// TwinCAT 3 PLC project MAIN
// ProgramVersion: 3.1.0.9
// CompilerDefines: VISU_USEWSTRING
// libraries:
//   VisuElem3DPath, 3.5.6.0 (System)
//   VisuElemMeter, 3.5.6.0 (System)
//   VisuElems, 3.5.6.10 (System)
//   VisuElemsDateTime, 3.5.6.0 (System)
//   VisuElemsSpecialControls, 3.5.6.0 (System)
//   VisuElemsWinControls, 3.5.6.0 (System)
//   VisuElemTextEditor, 3.5.6.0 (System)
//   visuinputs, 3.5.6.0 (system)
//   VisuNativeControl, 3.5.6.0 (System)
//   Tc2_MC2, * (Beckhoff Automation GmbH)
//   Tc2_NcFifoAxes, * (Beckhoff Automation GmbH)
//   Tc2_Standard, * (Beckhoff Automation GmbH)
//   Tc2_System, * (Beckhoff Automation GmbH)
//   Tc2_Utilities, * (Beckhoff Automation GmbH)
//   Tc3_Interfaces, * (Beckhoff Automation GmbH)
//   Tc3_Module, * (Beckhoff Automation GmbH)
//   VisuDialogs, * (System)
// project tree:
//   DUTs/ ST_CSV_Record.TcDUT
//   / GlobalTextList.TcGTLO, PlcTask.TcTTO, VISU_TASK.TcTTO, 视图管理器.TcVMO (not stored)
//   GVLs/ GVL.TcGVL
//   POUs/ AxisEnable.TcPOU (not stored), AxisMoveAbsoulte.TcPOU, AxisReset.TcPOU, AxisStop.TcPOU, Homing.TcPOU, MAIN.TcPOU, Move_JOG.TcPOU
//   POUs/CSV read_write in text mode/ P_TextModeRead.TcPOU, P_TextModeWrite.TcPOU
//   VISUs/ Visualization.TcVIS
// real-time tasks:
//   TASK PLC_TASK: cycle T#2ms, priority 20, ADS port 350
//   TASK VISU_TASK: cycle T#100000us, priority 30, ADS port 351
//   TASK Kine: cycle T#2ms, priority 21, ADS port 352
// motion (NC):
//   TASK NC-Task 1 SAF: cycle T#2ms, priority 4, ADS port 501
//   TASK NC-Task 1 SVB: cycle T#2ms, priority 8, ADS port 511
//   AXIS Axis 1 (id 1)
//     Dynamic: Acceleration=24000, Deceleration=24000, Jerk=96000
//     Velo: Maximum=6000
//     PositionAreaControl: Enable=false, RefSearch=false
//     TargetPosControl: Enable=false
//     OtherSettings: AllowMotionCmdToSlave=true
//     encoder EncType=19
//       EncPara: ScaleFactorNumerator=0.00274658203125, MaxCount=#xffffffff
//     drive DrvType=16
//       DrvPara: MaxCount=#xffffffff
//         Analog: VeloReferenz=6000
//         TimeComp: TaskDelayCycles=1
//     controller CtrType=1
//       CtrPara: PriorControlFactor=1
//         PosDiffControl: Enable=false
//         Observer: BandWidth=20
//   AXIS Axis 2 (id 2)
//     Dynamic: Acceleration=24000, Deceleration=24000, Jerk=96000
//     Velo: Maximum=6000
//     PositionAreaControl: Enable=false, RefSearch=false
//     TargetPosControl: Enable=false
//     OtherSettings: AllowMotionCmdToSlave=true
//     encoder EncType=19
//       EncPara: ScaleFactorNumerator=0.00274658203125, MaxCount=#xffffffff
//     drive DrvType=16
//       DrvPara: MaxCount=#xffffffff
//         Analog: VeloReferenz=6000
//         TimeComp: TaskDelayCycles=1
//     controller CtrType=1
//       CtrPara: PriorControlFactor=1
//         PosDiffControl: Enable=false
//         Observer: BandWidth=20
//   AXIS Axis 3 (id 3)
//     Dynamic: Acceleration=24000, Deceleration=24000, Jerk=96000
//     Velo: Maximum=6000
//     PositionAreaControl: Enable=false, RefSearch=false
//     TargetPosControl: Enable=false
//     OtherSettings: AllowMotionCmdToSlave=true
//     encoder EncType=19
//       EncPara: ScaleFactorNumerator=0.00274658203125, MaxCount=#xffffffff
//     drive DrvType=16
//       DrvPara: MaxCount=#xffffffff
//         Analog: VeloReferenz=6000
//         TimeComp: TaskDelayCycles=1
//     controller CtrType=1
//       CtrPara: PriorControlFactor=1
//         PosDiffControl: Enable=false
//         Observer: BandWidth=20
//   AXIS Axis 4 (id 4)
//     Dynamic: Acceleration=24000, Deceleration=24000, Jerk=96000
//     Velo: Maximum=6000
//     PositionAreaControl: Enable=false, RefSearch=false
//     TargetPosControl: Enable=false
//     OtherSettings: AllowMotionCmdToSlave=true
//     encoder EncType=19
//       EncPara: ScaleFactorNumerator=0.00274658203125, MaxCount=#xffffffff
//     drive DrvType=16
//       DrvPara: MaxCount=#xffffffff
//         Analog: VeloReferenz=6000
//         TimeComp: TaskDelayCycles=1
//     controller CtrType=1
//       CtrPara: PriorControlFactor=1
//         PosDiffControl: Enable=false
//         Observer: BandWidth=20
//   AXIS Axis 5 (id 5)
//     Dynamic: Acceleration=24000, Deceleration=24000, Jerk=96000
//     Velo: Maximum=6000
//     PositionAreaControl: Enable=false, RefSearch=false
//     TargetPosControl: Enable=false
//     OtherSettings: AllowMotionCmdToSlave=true
//     encoder EncType=19
//       EncPara: ScaleFactorNumerator=0.00274658203125, MaxCount=#xffffffff
//     drive DrvType=16
//       DrvPara: MaxCount=#xffffffff
//         Analog: VeloReferenz=6000
//         TimeComp: TaskDelayCycles=1
//     controller CtrType=1
//       CtrPara: PriorControlFactor=1
//         PosDiffControl: Enable=false
//         Observer: BandWidth=20
//   AXIS Axis 6 (id 6)
//     Dynamic: Acceleration=24000, Deceleration=24000, Jerk=96000
//     Velo: Maximum=6000
//     PositionAreaControl: Enable=false, RefSearch=false
//     TargetPosControl: Enable=false
//     OtherSettings: AllowMotionCmdToSlave=true
//     encoder EncType=19
//       EncPara: ScaleFactorNumerator=0.00274658203125, MaxCount=#xffffffff
//     drive DrvType=16
//       DrvPara: MaxCount=#xffffffff
//         Analog: VeloReferenz=6000
//         TimeComp: TaskDelayCycles=1
//     controller CtrType=1
//       CtrPara: PriorControlFactor=1
//         PosDiffControl: Enable=false
//         Observer: BandWidth=20
// I/O:
//   DEVICE Device 2 (EtherCAT), AmsNetId 192.168.1.1.3.1
//     Box 1 (TOYO NEC-100 Communicator) [TOYO NEC-100 Communicator]
//     Drive 2 (LAN9252-EVB-HBI) [LAN9252-EVB-HBI]
//       modules: Module 1 (csp - axis), Module 2 (csp - axis), Module 3 (csp - axis), Module 4 (csp - axis), Module 5 (csp - axis), Module 6 (csp - axis)
// variable links:
//   NC-Task 1 SAF/Axes/Axis 1 <-> Device 2 (EtherCAT)/Drive 2 (LAN9252-EVB-HBI)
//     Drive/Inputs/In/nState1 <-> Module 6 (csp - axis)/Inputs/Status Word
//     Drive/Inputs/In/nState2 <-> Module 6 (csp - axis)/Inputs/Status Word @bit 8
//     Drive/Outputs/Out/nCtrl1 <-> Module 6 (csp - axis)/Outputs/Control Word
//     Drive/Outputs/Out/nCtrl2 <-> Module 6 (csp - axis)/Outputs/Control Word @bit 8
//     Drive/Outputs/Out/nDataOut1 <-> Module 6 (csp - axis)/Outputs/TargetPosition
//     Enc/Inputs/In/nDataIn1 <-> Module 6 (csp - axis)/Inputs/ActualPosition
//     Enc/Inputs/In/nDcInputTime <-> InfoData/DcInputShift
//   NC-Task 1 SAF/Axes/Axis 2 <-> Device 2 (EtherCAT)/Drive 2 (LAN9252-EVB-HBI)
//     Drive/Inputs/In/nState1 <-> Module 2 (csp - axis)/Inputs/Status Word
//     Drive/Inputs/In/nState2 <-> Module 2 (csp - axis)/Inputs/Status Word @bit 8
//     Drive/Outputs/Out/nCtrl1 <-> Module 2 (csp - axis)/Outputs/Control Word
//     Drive/Outputs/Out/nCtrl2 <-> Module 2 (csp - axis)/Outputs/Control Word @bit 8
//     Drive/Outputs/Out/nDataOut1 <-> Module 2 (csp - axis)/Outputs/TargetPosition
//     Enc/Inputs/In/nDataIn1 <-> Module 2 (csp - axis)/Inputs/ActualPosition
//     Enc/Inputs/In/nDcInputTime <-> InfoData/DcInputShift
//   NC-Task 1 SAF/Axes/Axis 3 <-> Device 2 (EtherCAT)/Drive 2 (LAN9252-EVB-HBI)
//     Drive/Inputs/In/nState1 <-> Module 3 (csp - axis)/Inputs/Status Word
//     Drive/Inputs/In/nState2 <-> Module 3 (csp - axis)/Inputs/Status Word @bit 8
//     Drive/Outputs/Out/nCtrl1 <-> Module 3 (csp - axis)/Outputs/Control Word
//     Drive/Outputs/Out/nCtrl2 <-> Module 3 (csp - axis)/Outputs/Control Word @bit 8
//     Drive/Outputs/Out/nDataOut1 <-> Module 3 (csp - axis)/Outputs/TargetPosition
//     Enc/Inputs/In/nDataIn1 <-> Module 3 (csp - axis)/Inputs/ActualPosition
//     Enc/Inputs/In/nDcInputTime <-> InfoData/DcInputShift
//   NC-Task 1 SAF/Axes/Axis 4 <-> Device 2 (EtherCAT)/Drive 2 (LAN9252-EVB-HBI)
//     Drive/Inputs/In/nState1 <-> Module 4 (csp - axis)/Inputs/Status Word
//     Drive/Inputs/In/nState2 <-> Module 4 (csp - axis)/Inputs/Status Word @bit 8
//     Drive/Outputs/Out/nCtrl1 <-> Module 4 (csp - axis)/Outputs/Control Word
//     Drive/Outputs/Out/nCtrl2 <-> Module 4 (csp - axis)/Outputs/Control Word @bit 8
//     Drive/Outputs/Out/nDataOut1 <-> Module 4 (csp - axis)/Outputs/TargetPosition
//     Enc/Inputs/In/nDataIn1 <-> Module 4 (csp - axis)/Inputs/ActualPosition
//     Enc/Inputs/In/nDcInputTime <-> InfoData/DcInputShift
//   NC-Task 1 SAF/Axes/Axis 5 <-> Device 2 (EtherCAT)/Drive 2 (LAN9252-EVB-HBI)
//     Drive/Inputs/In/nDcOutputTime <-> InfoData/DcOutputShift
//     Drive/Inputs/In/nState1 <-> Module 5 (csp - axis)/Inputs/Status Word
//     Drive/Inputs/In/nState2 <-> Module 5 (csp - axis)/Inputs/Status Word @bit 8
//     Drive/Inputs/In/nState4 @bit 1 <-> WcState/InputToggle
//     Drive/Inputs/In/nState4 <-> WcState/WcState
//     Drive/Outputs/Out/nCtrl1 <-> Module 5 (csp - axis)/Outputs/Control Word
//     Drive/Outputs/Out/nCtrl2 <-> Module 5 (csp - axis)/Outputs/Control Word @bit 8
//     Drive/Outputs/Out/nDataOut1 <-> Module 5 (csp - axis)/Outputs/TargetPosition
//     Enc/Inputs/In/nDataIn1 <-> Module 5 (csp - axis)/Inputs/ActualPosition
//     Enc/Inputs/In/nDcInputTime <-> InfoData/DcInputShift
//     Enc/Inputs/In/nState4 @bit 1 <-> WcState/InputToggle
//     Enc/Inputs/In/nState4 <-> WcState/WcState
//   NC-Task 1 SAF/Axes/Axis 6 <-> Device 2 (EtherCAT)/Drive 2 (LAN9252-EVB-HBI)
//     Drive/Inputs/In/nState1 <-> Module 1 (csp - axis)/Inputs/Status Word
//     Drive/Inputs/In/nState2 <-> Module 1 (csp - axis)/Inputs/Status Word @bit 8
//     Drive/Outputs/Out/nCtrl1 <-> Module 1 (csp - axis)/Outputs/Control Word
//     Drive/Outputs/Out/nCtrl2 <-> Module 1 (csp - axis)/Outputs/Control Word @bit 8
//     Drive/Outputs/Out/nDataOut1 <-> Module 1 (csp - axis)/Outputs/TargetPosition
//     Enc/Inputs/In/nDataIn1 <-> Module 1 (csp - axis)/Inputs/ActualPosition
//     Enc/Inputs/In/nDcInputTime <-> InfoData/DcInputShift
//   MAIN/MAIN Instance <-> Device 2 (EtherCAT)/Box 1 (TOYO NEC-100 Communicator)
//     PlcTask Inputs/MAIN.EcdPos <-> TxPDO/Sa1/EcdPos
//     PlcTask Inputs/MAIN.Status <-> TxPDO/Sa1/Status
//     PlcTask Outputs/MAIN.ABSamount <-> RxPDO/Sa1/ABSamount
//     PlcTask Outputs/MAIN.Control <-> RxPDO/Sa1/Control
//     PlcTask Outputs/MAIN.MovType <-> RxPDO/Sa1/MovType
//   MAIN/MAIN Instance <-> NC-Task 1 SAF/Axes/Axis 1
//     PlcTask Inputs/GVL.Axis[0].NcToPlc <-> Outputs/ToPlc
//     PlcTask Outputs/GVL.Axis[0].PlcToNc <-> Inputs/FromPlc
//   MAIN/MAIN Instance <-> NC-Task 1 SAF/Axes/Axis 2
//     PlcTask Inputs/GVL.Axis[1].NcToPlc <-> Outputs/ToPlc
//     PlcTask Outputs/GVL.Axis[1].PlcToNc <-> Inputs/FromPlc
//   MAIN/MAIN Instance <-> NC-Task 1 SAF/Axes/Axis 3
//     PlcTask Inputs/GVL.Axis[2].NcToPlc <-> Outputs/ToPlc
//     PlcTask Outputs/GVL.Axis[2].PlcToNc <-> Inputs/FromPlc
//   MAIN/MAIN Instance <-> NC-Task 1 SAF/Axes/Axis 4
//     PlcTask Inputs/GVL.Axis[3].NcToPlc <-> Outputs/ToPlc
//     PlcTask Outputs/GVL.Axis[3].PlcToNc <-> Inputs/FromPlc
//   MAIN/MAIN Instance <-> NC-Task 1 SAF/Axes/Axis 5
//     PlcTask Inputs/GVL.Axis[4].NcToPlc <-> Outputs/ToPlc
//     PlcTask Outputs/GVL.Axis[4].PlcToNc <-> Inputs/FromPlc
//   MAIN/MAIN Instance <-> NC-Task 1 SAF/Axes/Axis 6
//     PlcTask Inputs/GVL.Axis[5].NcToPlc <-> Outputs/ToPlc
//     PlcTask Outputs/GVL.Axis[5].PlcToNc <-> Inputs/FromPlc
//   MAIN/MAIN Instance <-> Kinematic/Kinematic_Obj1 (CKineModule)
//     PlcTask Inputs/GVL.ExtPosOK <-> Outputs/ExtPosOK
//     PlcTask Inputs/GVL.ExtPosReady <-> Outputs/ExtPosReady
//     PlcTask Inputs/GVL.ExtPos[{0..5}] <-> Outputs/OutAngle[{0..5}]  (6 links)
//     PlcTask Inputs/GVL.Pos_Now[0] <-> Outputs/Pos_Now[0]
//     PlcTask Inputs/GVL.Pos_Now[1] <-> Outputs/Pos_Now[1]
//     PlcTask Inputs/GVL.Pos_Now[2] <-> Outputs/Pos_Now[2]
//     PlcTask Outputs/GVL.CMoveSpeed <-> Inputs/CSpeed
//     PlcTask Outputs/GVL.KineModuleJob <-> Inputs/KineModlueJob
//     PlcTask Outputs/GVL.LineMoveSpeed <-> Inputs/LineSpeed
//     PlcTask Outputs/GVL.OutActPos[{0..5}] <-> Inputs/InAngle[{5..0}]  (6 links)
//     PlcTask Outputs/GVL.OutCMovePos[0] <-> Inputs/CPos[0]
//     PlcTask Outputs/GVL.OutCMovePos[1] <-> Inputs/CPos[1]
//     PlcTask Outputs/GVL.OutCMovePos[2] <-> Inputs/CPos[2]
//     PlcTask Outputs/GVL.OutMovePos[0] <-> Inputs/InPos[0]
//     PlcTask Outputs/GVL.OutMovePos[1] <-> Inputs/InPos[1]
//     PlcTask Outputs/GVL.OutMovePos[2] <-> Inputs/InPos[2]

CONFIGURATION MAIN
    RESOURCE PLC ON TwinCAT3
        TASK PlcTask(INTERVAL := T#2ms, PRIORITY := 20);
        TASK VISU_TASK(INTERVAL := T#100000us, PRIORITY := 30);
        PROGRAM MAIN WITH PlcTask : MAIN;
        PROGRAM VisuElems_Visu_Prg WITH VISU_TASK : VisuElems.Visu_Prg;
    END_RESOURCE
END_CONFIGURATION

// ---- DUTs/ST_CSV_Record.TcDUT
TYPE ST_CSV_Record :
STRUCT
	sName 	: T_MaxString 	:= '';
	nNumber	: UDINT 		:= 0;
	fPos	: LREAL 		:= 0.0;
	bOP		: BOOL 			:= FALSE;
	sDesc	: STRING(40)	:= '';
	data	: ARRAY[0..7] OF BYTE;
END_STRUCT
END_TYPE

// ---- GVLs/GVL.TcGVL
VAR_GLOBAL CONSTANT
	MAX_CSV_ROWS 			: UDINT := 1;//1680;//hang
	MAX_CSV_COLUMNS 		: UDINT := 3;//lie 0-5
	MAX_CSV_FIELD_LENGTH	: UDINT := 20;
END_VAR

VAR_GLOBAL

axisNum: INT:=0;
//Axis Bind link
Axis:ARRAY[0..5]OF AXIS_REF;	

//Axis Power On
AxisPower:ARRAY[0..5]OF MC_Power;
AxisPowerTrigger:ARRAY[0..5]OF BOOL;
AxisPowerReady:ARRAY[0..5]OF BOOL;
AxisPowerBusy:ARRAY[0..5]OF BOOL;
AxisPowerActive:ARRAY[0..5]OF BOOL;
AxisPowerError:ARRAY[0..5]OF BOOL;
AxisPowerErrorID:ARRAY[0..5]OF UDINT;

//Axis Move Absolute
AxisMoveAbsolute:ARRAY[0..5]OF MC_MoveAbsolute;
AxisMoveTrigger:ARRAY[0..5]OF BOOL;
AxisMovePosition:ARRAY[0..5]OF LREAL;
AxisMoveSpeed:ARRAY[0..5]OF LREAL;
AxisMoveAcceleration:ARRAY[0..5]OF LREAL;
AxisMoveDeceleration:ARRAY[0..5]OF LREAL;
AxisMoveJerk:ARRAY[0..5]OF LREAL;
AxisMoveAbsoluteDone:ARRAY[0..5]OF BOOL;
AxisMoveAbsoluteBusy:ARRAY[0..5]OF BOOL;
AxisMoveAbsoluteActive:ARRAY[0..5]OF BOOL;
AxisMoveAbsoluteCommandAborted:ARRAY[0..5]OF BOOL;
AxisMoveAbsoluteError:ARRAY[0..5]OF BOOL;
AxisMoveAbsoluteErrorID:ARRAY[0..5]OF UDINT;

//Axis Stop
MC_Stop1:ARRAY[0..5]OF MC_Stop;
AxisStopTrigger:ARRAY[0..5]OF BOOL;
AxisStopDeceleration:ARRAY[0..5]OF LREAL;
AxisStopJerk:ARRAY[0..5]OF LREAL;
AxisStopDone:ARRAY[0..5]OF BOOL;
AxisStopBusy:ARRAY[0..5]OF BOOL;
AxisStopActive:ARRAY[0..5]OF BOOL;
AxisStopCommandAborted:ARRAY[0..5]OF BOOL;
AxisStopError:ARRAY[0..5]OF BOOL;
AxisStopErrorID:ARRAY[0..5]OF UDINT;

//MoveJOG
MoveJOG:ARRAY[0..5]OF MC_Jog;
JogFw:ARRAY[0..5]OF BOOL;
JogBw:ARRAY[0..5]OF BOOL;
JogMode:ARRAY[0..5]OF E_JogMode;
JogPosition:ARRAY[0..5]OF LREAL;
Jogvelocity:ARRAY[0..5]OF LREAL;
JogAcceleration:ARRAY[0..5]OF LREAL;
JogDeceleration:ARRAY[0..5]OF LREAL;
JogJerk:ARRAY[0..5]OF LREAL;
JogDone:ARRAY[0..5]OF BOOL;
JogBusy:ARRAY[0..5]OF BOOL;
JogActive:ARRAY[0..5]OF BOOL;
JogCommandAborted:ARRAY[0..5]OF BOOL;
JogError:ARRAY[0..5]OF BOOL;
JogErrorID:ARRAY[0..5]OF UDINT;

//Reset
MC_Resrt_0: ARRAY[0..5] OF MC_Reset;
AxisResetDone: ARRAY[0..5] OF BOOL;
AxisResetTrigger: ARRAY[0..5] OF BOOL;
AxisResetBusy: ARRAY[0..5] OF BOOL;
AxisResetError: ARRAY[0..5] OF BOOL;
AxisResetErrorID: ARRAY[0..5] OF UDINT;

//HOME
home_1: ARRAY[0..5] OF MC_HOME;
Home_Done: ARRAY[0..5] OF BOOL;
Home: ARRAY[0..5] OF BOOL;
Home_Pos: ARRAY[0..5] OF LREAL;
Home_Mode: ARRAY[0..5] OF MC_HomingMode;
Home_cal: ARRAY[0..5] OF BOOL;
Home_busy: ARRAY[0..5] OF BOOL;
Home_Active: ARRAY[0..5] OF BOOL;
Home_CommandAborted: ARRAY[0..5] OF BOOL;
Home_Error: ARRAY[0..5] OF BOOL;
Home_ErrorID: ARRAY[0..5] OF UDINT;
	
MoveA:ARRAY [0..5] OF LREAL;
MoveAString:ARRAY [0..5] OF STRING := ['0','0','0','0','0','0'];

FIFO_POS AT%I*:ARRAY[0..5]OF LREAL;//来自ros的外部位置
ExtPos AT%I*:ARRAY[0..5]OF LREAL;//来自CPPModule的外部位置
ExtPosOK AT%I*:BOOL;//外部位置执行结束标志
ExtPosReady AT%I*:BOOL;//外部位置规划完成
OutActPos AT%Q*:ARRAY[0..5]OF LREAL;//给CPPModule的实时位置

OutMovePos AT%Q*:ARRAY[0..2]OF LREAL;//直线规划增量
OutMovePosString:ARRAY[0..2]OF STRING := ['0','0','-0.1'];//增量字符串值
LineMoveSpeed AT%Q*:LREAL;//运动速度
LineMoveSpeedString:STRING:='0.05';

OutCMovePos AT%Q*:ARRAY[0..2]OF LREAL;//笛卡尔规划增量
OutCMovePosString:ARRAY[0..2]OF STRING := ['0.4','0.2','0.2'];//增量字符串值
CMoveSpeed AT%Q*:LREAL;//运动速度
CMoveSpeedString:STRING:='0.3';

KineModuleJob AT%Q*:INT:=0;//CPPModule状态机控制
Pos_Now AT%I*:ARRAY[0..2]OF LREAL;//CPPModule输出实时笛卡尔坐标
END_VAR

// ---- POUs/MAIN.TcPOU
PROGRAM MAIN
VAR
bChangeSeparatorToComma	: BOOL := TRUE;
P_TextModeWrite_WriteTrigger:BOOL:=FALSE;
P_TextModeWrite_WriteFilePath:T_MaxString := 'C:\Users\Administrator\Desktop\Pos.csv';
P_TextModeRead_ReadTrigger:BOOL:=FALSE;
P_TextModeRead_ReadFilePath:T_MaxString := 'C:\Users\Administrator\Desktop\Pos.csv';

CurrentJob: INT:= 0;//Job Code
CurrentJobState:STRING(80);//Say in which state

LAMP:BOOL;
POWER:BOOL;
Move_AB:BOOL;

SetPointGenEnable:ARRAY [0..5] OF MC_ExtSetPointGenEnable;
SetpointGenDisable:ARRAY [0..5] OF MC_ExtSetpointGenDisable;
SetPointGenEnable_output: ARRAY [0..5] OF ST_McOutputs;
SetPointGenDisable_output: ARRAY [0..5] OF ST_McOutputs;
enable:ARRAY [0..5] OF BOOL;
disable:ARRAY [0..5] OF BOOL;

position:ARRAY [0..5] OF LREAL;
velocity:ARRAY [0..5] OF LREAL;
direction:ARRAY [0..5] OF DINT;
acceleration:ARRAY [0..5] OF LREAL;

Pos_arr1:ARRAY[0..4999,0..5] OF LREAL;
i:INT;
FiFo_GetDimension: FiFoGetDimension;
fifo_display: STRING(255);

FiFo_GroupIntegrate1,FiFo_GroupIntegrate2,FiFo_GroupIntegrate3,FiFo_GroupIntegrate4,FiFo_GroupIntegrate6,FiFo_GroupIntegrate5: FiFoGroupIntegrate;
FiFo_SetChannelOverride:FiFoSetChannelOverride;
FiFo_Groupout1,FiFo_Groupout2,FiFo_Groupout3,FiFo_Groupout4,FiFo_Groupout5,FiFo_Groupout6,FiFo_Disintegrate,FiFo_Override_output:st_mcoutputs;
integrate_do:BOOL;
FiFo_GroupDisintegrate:FiFoGroupDisintegrate;

FiFo_Start:FiFoStart;
start_do:BOOL;
FiFo_Stop:FiFoStop;
stop_do:BOOL;
fifo_startoutput,fifo_stopoutput:st_mcoutputs;

FiFo_Write:FiFoWrite;
FIFO_write_do:BOOL;
FiFo_overWrite:FiFoOverwrite;
FIFO_overwrite_do:BOOL;
FIFO_write_output:st_mcoutputs;

END_VAR
VAR CONSTANT
	GlobalSetSpeed : ARRAY[0..5]OF LREAL:=[3200,3200,3200,3200,3200,3200];
END_VAR

IF bChangeSeparatorToComma THEN
	DEFAULT_CSV_FIELD_SEP := 16#2C;(* Comma ASCII code *)
ELSE
	DEFAULT_CSV_FIELD_SEP := 16#3B;(* Semicolon ASCII code *)
END_IF

IF FiFo_GetDimension.iNoOfAxes=6 AND FiFo_GetDimension.iNoOfFifoEntries=200 THEN
	fifo_display:='Parameters OK';
ELSE
	fifo_display:='Parameters Bad';
END_IF

//fifo();

GVL.LineMoveSpeed:=STRING_TO_LREAL(GVL.LineMoveSpeedString);
GVL.CMoveSpeed:=STRING_TO_LREAL(GVL.CMoveSpeedString);
GVL.OutMovePos[0]:=STRING_TO_LREAL(GVL.OutMovePosString[0]);
GVL.OutMovePos[1]:=STRING_TO_LREAL(GVL.OutMovePosString[1]);
GVL.OutMovePos[2]:=STRING_TO_LREAL(GVL.OutMovePosString[2]);
GVL.OutCMovePos[0]:=STRING_TO_LREAL(GVL.OutCMovePosString[0]);
GVL.OutCMovePos[1]:=STRING_TO_LREAL(GVL.OutCMovePosString[1]);
GVL.OutCMovePos[2]:=STRING_TO_LREAL(GVL.OutCMovePosString[2]);
GVL.MoveA[0]:=STRING_TO_LREAL(GVL.MoveAString[0])*24.995;
GVL.MoveA[1]:=STRING_TO_LREAL(GVL.MoveAString[1])*32.28;
GVL.MoveA[2]:=STRING_TO_LREAL(GVL.MoveAString[2])*49.845;
GVL.MoveA[3]:=STRING_TO_LREAL(GVL.MoveAString[3])*50.905;
GVL.MoveA[4]:=STRING_TO_LREAL(GVL.MoveAString[4])*80.34;
GVL.MoveA[5]:=STRING_TO_LREAL(GVL.MoveAString[5])*60.5;
GVL.OutActPos[0]:=-GVL.Axis[0].NcToPlc.ActPos/24.995;
GVL.OutActPos[1]:=-GVL.Axis[1].NcToPlc.ActPos/32.28;
GVL.OutActPos[2]:=GVL.Axis[2].NcToPlc.ActPos/49.845;
GVL.OutActPos[3]:=GVL.Axis[3].NcToPlc.ActPos/50.905;
GVL.OutActPos[4]:=GVL.Axis[4].NcToPlc.ActPos/80.34;
GVL.OutActPos[5]:=GVL.Axis[5].NcToPlc.ActPos/60.5;

IF GVL.ExtPosReady = FALSE THEN	
MC_ExtSetPointGenFeed(Position:=-GVL.OutActPos[0]*24.995,Velocity:= 0,Acceleration:=0,Direction:=1,Axis:=Axis[0]);	
MC_ExtSetPointGenFeed(Position:=-GVL.OutActPos[1]*32.28,Velocity:= 0,Acceleration:=0,Direction:=1,Axis:=Axis[1]);		
MC_ExtSetPointGenFeed(Position:=GVL.OutActPos[2]*49.845,Velocity:= 0,Acceleration:=0,Direction:=1,Axis:=Axis[2]);		
MC_ExtSetPointGenFeed(Position:=GVL.OutActPos[3]*50.905,Velocity:= 0,Acceleration:=0,Direction:=1,Axis:=Axis[3]);		
MC_ExtSetPointGenFeed(Position:=GVL.OutActPos[4]*80.34,Velocity:= 0,Acceleration:=0,Direction:=1,Axis:=Axis[4]);		
MC_ExtSetPointGenFeed(Position:=GVL.OutActPos[5]*60.5,Velocity:= 0,Acceleration:=0,Direction:=1,Axis:=Axis[5]);		
END_IF

CASE CurrentJob OF	
	0://None state
		AxisStopTrigger[0]:=FALSE;AxisStopTrigger[1]:=FALSE;AxisStopTrigger[2]:=FALSE;
		AxisStopTrigger[3]:=FALSE;AxisStopTrigger[4]:=FALSE;AxisStopTrigger[5]:=FALSE;
		AxisStop();//失能功能块
		
		JogFw[0]:=FALSE;JogFw[1]:=FALSE;JogFw[2]:=FALSE;JogFw[3]:=FALSE;JogFw[4]:=FALSE;JogFw[5]:=FALSE;
		JogBw[0]:=FALSE;JogBw[1]:=FALSE;JogBw[2]:=FALSE;JogBw[3]:=FALSE;JogBw[4]:=FALSE;JogBw[5]:=FALSE;
		Move_JOG();//失能功能块
		
		AxisMoveTrigger[0]:=FALSE;AxisMoveTrigger[1]:=FALSE;AxisMoveTrigger[2]:=FALSE;
		AxisMoveTrigger[3]:=FALSE;AxisMoveTrigger[4]:=FALSE;AxisMoveTrigger[5]:=FALSE;
		AxisMoveAbsoulte();//失能功能块
		
		Home[0]:=FALSE;Home[1]:=FALSE;Home[2]:=FALSE;
		Home[3]:=FALSE;Home[4]:=FALSE;Home[5]:=FALSE;
		Homing();//失能功能块	

		AxisResetTrigger[0]:=FALSE;AxisResetTrigger[1]:=FALSE;AxisResetTrigger[2]:=FALSE;
		AxisResetTrigger[3]:=FALSE;AxisResetTrigger[4]:=FALSE;AxisResetTrigger[5]:=FALSE;
		AxisReset();//失能功能块
		
		P_TextModeWrite_WriteTrigger:=FALSE;
		P_TextModeWrite();	
		P_TextModeRead_ReadTrigger:=FALSE;
		P_TextModeRead();//失能功能块
		
		SetPointGenEnable[0].Execute:=FALSE;SetPointGenEnable[1].Execute:=FALSE;
		SetPointGenEnable[2].Execute:=FALSE;SetPointGenEnable[3].Execute:=FALSE;
		SetPointGenEnable[4].Execute:=FALSE;SetPointGenEnable[5].Execute:=FALSE;

		SetPointGenDisable[0].Execute:=FALSE;SetPointGenDisable[1].Execute:=FALSE;		
		SetPointGenDisable[2].Execute:=FALSE;SetPointGenDisable[3].Execute:=FALSE;		
		SetPointGenDisable[4].Execute:=FALSE;SetPointGenDisable[5].Execute:=FALSE;		
		setpositionGen();
		
		JogMode[0]:=MC_JOGMODE_STANDARD_FAST;
		JogMode[1]:=MC_JOGMODE_STANDARD_FAST;
		JogMode[2]:=MC_JOGMODE_STANDARD_FAST;
		JogMode[3]:=MC_JOGMODE_STANDARD_FAST;
		JogMode[4]:=MC_JOGMODE_STANDARD_FAST;
		JogMode[5]:=MC_JOGMODE_STANDARD_FAST;

		GVL.KineModuleJob:=0;
	
		CurrentJobState:='Wait Command';
		i:=0;
	1://SetZero
		Home[0]:=TRUE;Home[1]:=TRUE;Home[2]:=TRUE;
		Home[3]:=TRUE;Home[4]:=TRUE;Home[5]:=TRUE;
		Home_Mode[0]:=MC_Direct;Home_Mode[1]:=MC_Direct;Home_Mode[2]:=MC_Direct;
		Home_Mode[3]:=MC_Direct;Home_Mode[4]:=MC_Direct;Home_Mode[5]:=MC_Direct;
		Home_Pos[0]:=0;Home_Pos[1]:=0;Home_Pos[2]:=0;
		Home_Pos[3]:=0;Home_Pos[4]:=0;Home_Pos[5]:=0;
		Homing();

		IF Home_Done[0]=TRUE AND 
		   Home_Done[1]=TRUE AND 
		   Home_Done[2]=TRUE AND 
		   Home_Done[3]=TRUE AND 
		   Home_Done[4]=TRUE AND 
		   Home_Done[5]=TRUE THEN
			CurrentJob:=0;
			CurrentJobState:='Set Origin Done!';
		ELSE
			CurrentJobState:='Set Origin Doing';
		END_IF
	2://直线插补
		setpointgenenable[0].Execute:=TRUE;setpointgenenable[1].Execute:=TRUE;
		setpointgenenable[2].Execute:=TRUE;setpointgenenable[3].Execute:=TRUE;
		setpointgenenable[4].Execute:=TRUE;setpointgenenable[5].Execute:=TRUE;
		IF  SetPointGenEnable[0].Enabled AND
			SetPointGenEnable[1].Enabled AND
			SetPointGenEnable[2].Enabled AND
			SetPointGenEnable[3].Enabled AND
			SetPointGenEnable[4].Enabled AND
			SetPointGenEnable[5].Enabled THEN

			//IF(GVL.ExtPosOK = TRUE) THEN
			IF i > 4998 THEN
				SetPointGenDisable[0].Execute:=TRUE;SetPointGenDisable[1].Execute:=TRUE;
				SetPointGenDisable[2].Execute:=TRUE;SetPointGenDisable[3].Execute:=TRUE;
				SetPointGenDisable[4].Execute:=TRUE;SetPointGenDisable[5].Execute:=TRUE;
				setpositionGen();
				CurrentJob:=0;
			ELSE
				i:=i+1;
		
				MC_ExtSetPointGenFeed(Position:=Pos_arr1[i,0]*24.995,Velocity:= 0,Acceleration:=0,Direction:=1,Axis:=Axis[0]);
			
				MC_ExtSetPointGenFeed(Position:=Pos_arr1[i,1]*32.28,Velocity:= 0,Acceleration:=0,Direction:=1,Axis:=Axis[1]);
			
				MC_ExtSetPointGenFeed(Position:=Pos_arr1[i,2]*49.845,Velocity:= 0,Acceleration:=0,Direction:=1,Axis:=Axis[2]);
			
				MC_ExtSetPointGenFeed(Position:=Pos_arr1[i,3]*50.905,Velocity:= 0,Acceleration:=0,Direction:=1,Axis:=Axis[3]);
			
				MC_ExtSetPointGenFeed(Position:=Pos_arr1[i,4]*80.34,Velocity:= 0,Acceleration:=0,Direction:=1,Axis:=Axis[4]);
			
				MC_ExtSetPointGenFeed(Position:=Pos_arr1[i,5]*60.5,Velocity:= 0,Acceleration:=0,Direction:=1,Axis:=Axis[5]);
			END_IF
			//GVL.KineModuleJob:=4;
			//IF GVL.ExtPosReady THEN
			//MC_ExtSetPointGenFeed(Position:=-ExtPos[0]*24.995,Velocity:= 0,Acceleration:=0,Direction:=1,Axis:=Axis[0]);
			
			//MC_ExtSetPointGenFeed(Position:=-ExtPos[1]*32.28,Velocity:= 0,Acceleration:=0,Direction:=1,Axis:=Axis[1]);
			
			//MC_ExtSetPointGenFeed(Position:=ExtPos[2]*49.845,Velocity:= 0,Acceleration:=0,Direction:=1,Axis:=Axis[2]);
			
			//MC_ExtSetPointGenFeed(Position:=ExtPos[3]*50.905,Velocity:= 0,Acceleration:=0,Direction:=1,Axis:=Axis[3]);
			
			//MC_ExtSetPointGenFeed(Position:=ExtPos[4]*80.34,Velocity:= 0,Acceleration:=0,Direction:=1,Axis:=Axis[4]);
			
			//MC_ExtSetPointGenFeed(Position:=ExtPos[5]*60.5,Velocity:= 0,Acceleration:=0,Direction:=1,Axis:=Axis[5]);		
			//END_IF
		END_IF
		setpositionGen();
	3://JogForward
		JogFw[axisNum]:=TRUE;
		Move_JOG();
		CurrentJob:=3;
		CurrentJobState:='Jog Forward';
	4://JogBackward
		JogBw[axisNum]:=TRUE;
		Move_JOG();
		CurrentJob:=4;
		CurrentJobState:='Jog Backward';
	5://Stop
		AxisStopDeceleration[0]:=15000;AxisStopDeceleration[1]:=15000;AxisStopDeceleration[2]:=15000;
		AxisStopDeceleration[3]:=15000;AxisStopDeceleration[4]:=15000;AxisStopDeceleration[5]:=15000;
		AxisStopTrigger[0]:=TRUE;AxisStopTrigger[1]:=TRUE;AxisStopTrigger[2]:=TRUE;
		AxisStopTrigger[3]:=TRUE;AxisStopTrigger[4]:=TRUE;AxisStopTrigger[5]:=TRUE;
		AxisStop();
		IF AxisStopDone[0]=TRUE AND
		   AxisStopDone[1]=TRUE AND
		   AxisStopDone[2]=TRUE AND
		   AxisStopDone[3]=TRUE AND
		   AxisStopDone[4]=TRUE AND
		   AxisStopDone[5]=TRUE THEN
			CurrentJobState:='Stop Done';
			CurrentJob:=0;
		ELSE
			CurrentJobState:='Stop Doing';
		END_IF
	6://Move To HOME
		AxisMovePosition[0]:=-3683.8943;AxisMovePosition[1]:=5173.9531;AxisMovePosition[2]:=318.8809;
		AxisMovePosition[3]:=5194.3991;AxisMovePosition[4]:=307.0219;AxisMovePosition[5]:=774.2587;	
		AxisMoveSpeed[0]:=2000;AxisMoveSpeed[1]:=2000;AxisMoveSpeed[2]:=2000;
		AxisMoveSpeed[3]:=2000;AxisMoveSpeed[4]:=2000;AxisMoveSpeed[5]:=2000;
		
		AxisMoveTrigger[0]:=TRUE;AxisMoveTrigger[1]:=TRUE;AxisMoveTrigger[2]:=TRUE;
		AxisMoveTrigger[3]:=TRUE;AxisMoveTrigger[4]:=TRUE;AxisMoveTrigger[5]:=TRUE;
		AxisMoveAbsoulte();
		
		IF AxisMoveAbsoluteDone[0]=TRUE AND 
		   AxisMoveAbsoluteDone[1]=TRUE AND 
		   AxisMoveAbsoluteDone[2]=TRUE AND 
		   AxisMoveAbsoluteDone[3]=TRUE AND 
		   AxisMoveAbsoluteDone[4]=TRUE AND 
		   AxisMoveAbsoluteDone[5]=TRUE THEN			
			CurrentJobState:='Home Done';
			CurrentJob:=1;			
		ELSE
			CurrentJobState:='Home Doing';
		END_IF
	7://Move To A
		AxisMovePosition[0]:=MoveA[0];AxisMovePosition[1]:=MoveA[1];AxisMovePosition[2]:=MoveA[2];
		AxisMovePosition[3]:=MoveA[3];AxisMovePosition[4]:=MoveA[4];AxisMovePosition[5]:=MoveA[5];
		
		AxisMoveSpeed[0]:=GlobalSetSpeed[0];AxisMoveSpeed[1]:=GlobalSetSpeed[1];AxisMoveSpeed[2]:=GlobalSetSpeed[2];
		AxisMoveSpeed[3]:=GlobalSetSpeed[3];AxisMoveSpeed[4]:=GlobalSetSpeed[4];AxisMoveSpeed[5]:=GlobalSetSpeed[5];
		
		AxisMoveTrigger[0]:=TRUE;AxisMoveTrigger[1]:=TRUE;AxisMoveTrigger[2]:=TRUE;
		AxisMoveTrigger[3]:=TRUE;AxisMoveTrigger[4]:=TRUE;AxisMoveTrigger[5]:=TRUE;
		AxisMoveAbsoulte();
		
		IF AxisMoveAbsoluteDone[0]=TRUE AND 
		   AxisMoveAbsoluteDone[1]=TRUE AND 
		   AxisMoveAbsoluteDone[2]=TRUE AND 
		   AxisMoveAbsoluteDone[3]=TRUE AND 
		   AxisMoveAbsoluteDone[4]=TRUE AND 
		   AxisMoveAbsoluteDone[5]=TRUE THEN		
			CurrentJobState:='MOVE A Done';
			CurrentJob:=0;		
		ELSE
			CurrentJobState:='MOVE A Doing';
		END_IF
	8://往复运动
		IF Move_AB=FALSE THEN
		//AxisMovePosition[0]:=-742579.6646;AxisMovePosition[1]:=5125.997925;AxisMovePosition[2]:=223.8519;
		//AxisMovePosition[3]:=5161.5829;AxisMovePosition[4]:=-31.9675;AxisMovePosition[5]:=774.2587;	
		AxisMovePosition[0]:=0;AxisMovePosition[1]:=0;AxisMovePosition[2]:=0;
		AxisMovePosition[3]:=0;AxisMovePosition[4]:=0;AxisMovePosition[5]:=0;
		ELSE
		AxisMovePosition[0]:=MoveA[0];AxisMovePosition[1]:=MoveA[1];AxisMovePosition[2]:=MoveA[2];
		AxisMovePosition[3]:=MoveA[3];AxisMovePosition[4]:=MoveA[4];AxisMovePosition[5]:=MoveA[5];	
		END_IF
		AxisMoveSpeed[0]:=2000;AxisMoveSpeed[1]:=2000;AxisMoveSpeed[2]:=2000;
		AxisMoveSpeed[3]:=2000;AxisMoveSpeed[4]:=2000;AxisMoveSpeed[5]:=2000;
		
		AxisMoveTrigger[0]:=TRUE;AxisMoveTrigger[1]:=TRUE;AxisMoveTrigger[2]:=TRUE;
		AxisMoveTrigger[3]:=TRUE;AxisMoveTrigger[4]:=TRUE;AxisMoveTrigger[5]:=TRUE;
		AxisMoveAbsoulte();
		
		IF AxisMoveAbsoluteDone[0]=TRUE AND 
		   AxisMoveAbsoluteDone[1]=TRUE AND 
		   AxisMoveAbsoluteDone[2]=TRUE AND 
		   AxisMoveAbsoluteDone[3]=TRUE AND 
		   AxisMoveAbsoluteDone[4]=TRUE AND 
		   AxisMoveAbsoluteDone[5]=TRUE THEN	
		   Move_AB:= NOT Move_AB;
		   AxisMoveTrigger[0]:=FALSE;AxisMoveTrigger[1]:=FALSE;AxisMoveTrigger[2]:=FALSE;
		   AxisMoveTrigger[3]:=FALSE;AxisMoveTrigger[4]:=FALSE;AxisMoveTrigger[5]:=FALSE;
		   AxisMoveAbsoulte();//失能功能块
		END_IF
		CurrentJobState:='Reciprocating Doing';
	9://复位
		AxisResetTrigger[0]:=TRUE;AxisResetTrigger[1]:=TRUE;AxisResetTrigger[2]:=TRUE;
		AxisResetTrigger[3]:=TRUE;AxisResetTrigger[4]:=TRUE;AxisResetTrigger[5]:=TRUE;
		AxisReset();
		IF AxisResetDone[0]=TRUE AND
		   AxisResetDone[1]=TRUE AND
		   AxisResetDone[2]=TRUE AND
		   AxisResetDone[3]=TRUE AND
		   AxisResetDone[4]=TRUE AND
		   AxisResetDone[5]=TRUE THEN	
			CurrentJobState:='Axis Reset Done';
			CurrentJob:=0;
		ELSE
			CurrentJobState:='Axis Reset Doing';
		END_IF
	10://read csv
		//P_TextModeRead_ReadTrigger:=TRUE;
		//CurrentJobState:='Read CSV';
		//P_TextModeRead();
		GVL.KineModuleJob:=2;
		CurrentJob:=0;
	11://Move to origin
		AxisMovePosition[0]:=0;AxisMovePosition[1]:=0;AxisMovePosition[2]:=0;
		AxisMovePosition[3]:=0;AxisMovePosition[4]:=0;AxisMovePosition[5]:=0;
		
		AxisMoveSpeed[0]:=2000;AxisMoveSpeed[1]:=2000;AxisMoveSpeed[2]:=2000;
		AxisMoveSpeed[3]:=2000;AxisMoveSpeed[4]:=2000;AxisMoveSpeed[5]:=2000;
		
		AxisMoveTrigger[0]:=TRUE;AxisMoveTrigger[1]:=TRUE;AxisMoveTrigger[2]:=TRUE;
		AxisMoveTrigger[3]:=TRUE;AxisMoveTrigger[4]:=TRUE;AxisMoveTrigger[5]:=TRUE;
		AxisMoveAbsoulte();
		
		IF AxisMoveAbsoluteDone[0]=TRUE AND 
		   AxisMoveAbsoluteDone[1]=TRUE AND 
		   AxisMoveAbsoluteDone[2]=TRUE AND 
		   AxisMoveAbsoluteDone[3]=TRUE AND 
		   AxisMoveAbsoluteDone[4]=TRUE AND 
		   AxisMoveAbsoluteDone[5]=TRUE THEN		
			CurrentJobState:='MOVE Origin Done';
			CurrentJob:=0;		
		ELSE
			CurrentJobState:='MOVE Origin Doing';
		END_IF
	12://直线插补
		setpointgenenable[0].Execute:=TRUE;setpointgenenable[1].Execute:=TRUE;
		setpointgenenable[2].Execute:=TRUE;setpointgenenable[3].Execute:=TRUE;
		setpointgenenable[4].Execute:=TRUE;setpointgenenable[5].Execute:=TRUE;
		IF  SetPointGenEnable[0].Enabled AND
			SetPointGenEnable[1].Enabled AND
			SetPointGenEnable[2].Enabled AND
			SetPointGenEnable[3].Enabled AND
			SetPointGenEnable[4].Enabled AND
			SetPointGenEnable[5].Enabled THEN
			
			IF(GVL.ExtPosOK = TRUE) THEN			
				SetPointGenDisable[0].Execute:=TRUE;SetPointGenDisable[1].Execute:=TRUE;
				SetPointGenDisable[2].Execute:=TRUE;SetPointGenDisable[3].Execute:=TRUE;
				SetPointGenDisable[4].Execute:=TRUE;SetPointGenDisable[5].Execute:=TRUE;
				setpositionGen();
				CurrentJob:=0;
			END_IF
			
			GVL.KineModuleJob:=3;
			IF GVL.ExtPosReady THEN
			MC_ExtSetPointGenFeed(Position:=ExtPos[0]*24.995,Velocity:= 0,Acceleration:=0,Direction:=1,Axis:=Axis[0]);
			
			MC_ExtSetPointGenFeed(Position:=-ExtPos[1]*32.28,Velocity:= 0,Acceleration:=0,Direction:=1,Axis:=Axis[1]);
			
			MC_ExtSetPointGenFeed(Position:=ExtPos[2]*49.845,Velocity:= 0,Acceleration:=0,Direction:=1,Axis:=Axis[2]);
			
			MC_ExtSetPointGenFeed(Position:=ExtPos[3]*50.905,Velocity:= 0,Acceleration:=0,Direction:=1,Axis:=Axis[3]);
			
			MC_ExtSetPointGenFeed(Position:=ExtPos[4]*80.34,Velocity:= 0,Acceleration:=0,Direction:=1,Axis:=Axis[4]);
			
			MC_ExtSetPointGenFeed(Position:=ExtPos[5]*60.5,Velocity:= 0,Acceleration:=0,Direction:=1,Axis:=Axis[5]);		
			END_IF
		END_IF
		setpositionGen();
	13://关节空间运动
		GVL.KineModuleJob:=1;
		CurrentJob:=0;
END_CASE

//错误检测
IF  AxisPowerError[0] OR
	AxisPowerError[1] OR
	AxisPowerError[2] OR
	AxisPowerError[3] OR
	AxisPowerError[4] OR
	AxisPowerError[5] THEN
	//POWER:=FALSE;
	CurrentJob:=9;
END_IF
//电机上下电
IF POWER=TRUE THEN
	AxisPowerTrigger[0]:=TRUE;
	AxisPowerTrigger[1]:=TRUE;
	AxisPowerTrigger[2]:=TRUE;
	AxisPowerTrigger[3]:=TRUE;
	AxisPowerTrigger[4]:=TRUE;
	AxisPowerTrigger[5]:=TRUE;
	AxisEnable();
	IF  AxisPowerReady[0]=TRUE AND 
		AxisPowerReady[1]=TRUE AND 
		AxisPowerReady[2]=TRUE AND 
		AxisPowerReady[3]=TRUE AND
		AxisPowerReady[4]=TRUE AND 
		AxisPowerReady[5]=TRUE THEN
		LAMP:=TRUE;
	END_IF
ELSE
	AxisPowerTrigger[0]:=FALSE;
	AxisPowerTrigger[1]:=FALSE;
	AxisPowerTrigger[2]:=FALSE;
	AxisPowerTrigger[3]:=FALSE;
	AxisPowerTrigger[4]:=FALSE;
	AxisPowerTrigger[5]:=FALSE;
	AxisEnable();
	IF  AxisPowerReady[0]=FALSE AND
		AxisPowerReady[1]=FALSE AND
		AxisPowerReady[2]=FALSE AND
		AxisPowerReady[3]=FALSE AND
		AxisPowerReady[4]=FALSE AND
		AxisPowerReady[5]=FALSE THEN
		LAMP:=FALSE;   
	END_IF
END_IF

ACTION fifo:
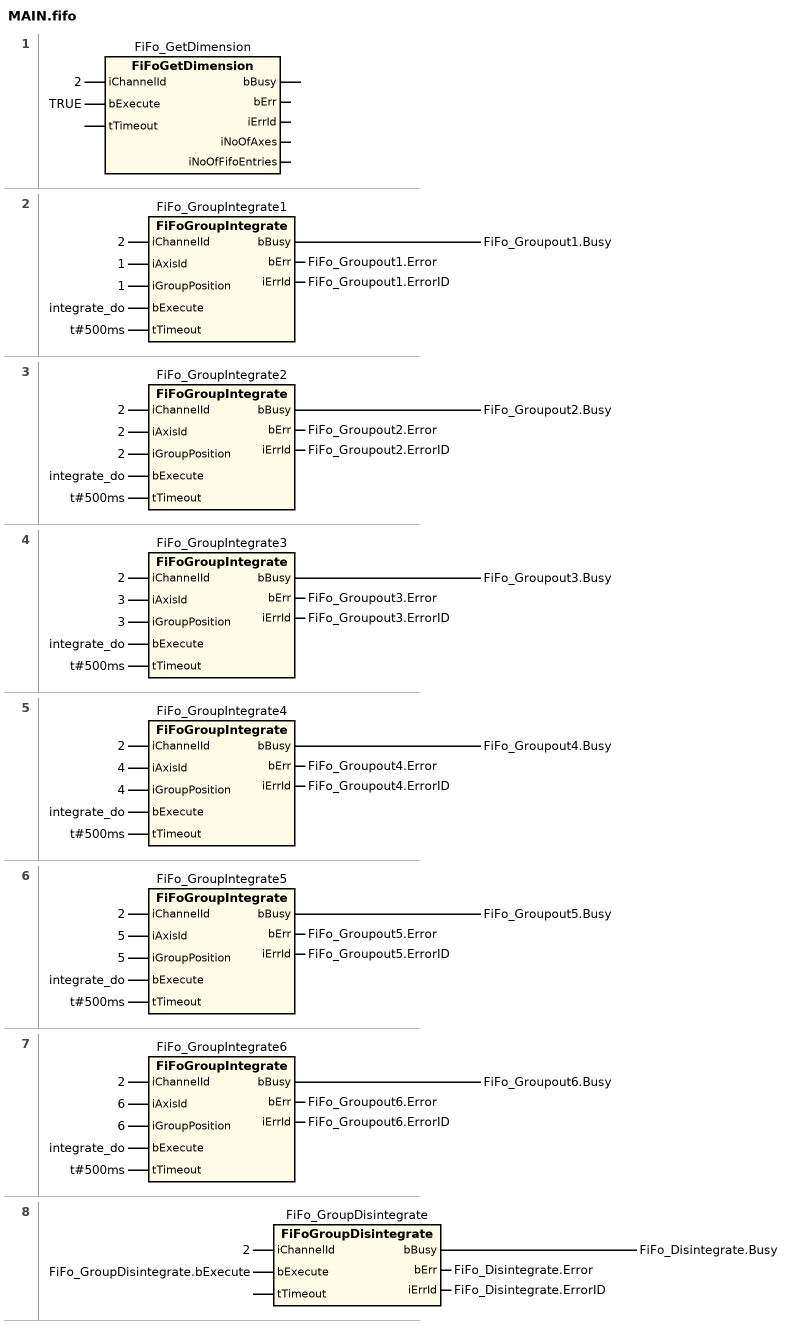
// NETWORK 1
FiFo_GetDimension(iChannelId := 2, bExecute := TRUE); // FiFoGetDimension

// NETWORK 2
FiFo_GroupIntegrate1(
    iChannelId := 2,
    iAxisId := 1,
    iGroupPosition := 1,
    bExecute := integrate_do,
    tTimeout := t#500ms,
    bErr => FiFo_Groupout1.Error,
    iErrId => FiFo_Groupout1.ErrorID); // FiFoGroupIntegrate
FiFo_Groupout1.Busy := FiFo_GroupIntegrate1.bBusy;

// NETWORK 3
FiFo_GroupIntegrate2(
    iChannelId := 2,
    iAxisId := 2,
    iGroupPosition := 2,
    bExecute := integrate_do,
    tTimeout := t#500ms,
    bErr => FiFo_Groupout2.Error,
    iErrId => FiFo_Groupout2.ErrorID); // FiFoGroupIntegrate
FiFo_Groupout2.Busy := FiFo_GroupIntegrate2.bBusy;

// NETWORK 4
FiFo_GroupIntegrate3(
    iChannelId := 2,
    iAxisId := 3,
    iGroupPosition := 3,
    bExecute := integrate_do,
    tTimeout := t#500ms,
    bErr => FiFo_Groupout3.Error,
    iErrId => FiFo_Groupout3.ErrorID); // FiFoGroupIntegrate
FiFo_Groupout3.Busy := FiFo_GroupIntegrate3.bBusy;

// NETWORK 5
FiFo_GroupIntegrate4(
    iChannelId := 2,
    iAxisId := 4,
    iGroupPosition := 4,
    bExecute := integrate_do,
    tTimeout := t#500ms,
    bErr => FiFo_Groupout4.Error,
    iErrId => FiFo_Groupout4.ErrorID); // FiFoGroupIntegrate
FiFo_Groupout4.Busy := FiFo_GroupIntegrate4.bBusy;

// NETWORK 6
FiFo_GroupIntegrate5(
    iChannelId := 2,
    iAxisId := 5,
    iGroupPosition := 5,
    bExecute := integrate_do,
    tTimeout := t#500ms,
    bErr => FiFo_Groupout5.Error,
    iErrId => FiFo_Groupout5.ErrorID); // FiFoGroupIntegrate
FiFo_Groupout5.Busy := FiFo_GroupIntegrate5.bBusy;

// NETWORK 7
FiFo_GroupIntegrate6(
    iChannelId := 2,
    iAxisId := 6,
    iGroupPosition := 6,
    bExecute := integrate_do,
    tTimeout := t#500ms,
    bErr => FiFo_Groupout6.Error,
    iErrId => FiFo_Groupout6.ErrorID); // FiFoGroupIntegrate
FiFo_Groupout6.Busy := FiFo_GroupIntegrate6.bBusy;

// NETWORK 8
FiFo_GroupDisintegrate(
    iChannelId := 2,
    bExecute := FiFo_GroupDisintegrate.bExecute,
    bErr => FiFo_Disintegrate.Error,
    iErrId => FiFo_Disintegrate.ErrorID); // FiFoGroupDisintegrate
FiFo_Disintegrate.Busy := FiFo_GroupDisintegrate.bBusy;

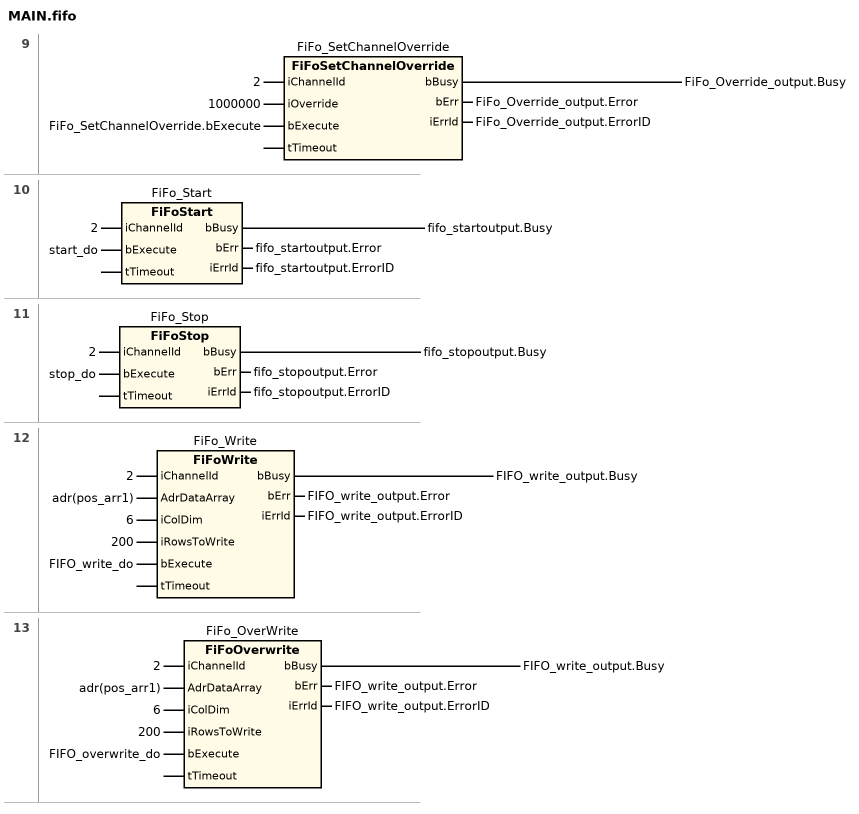
// NETWORK 9
FiFo_SetChannelOverride(
    iChannelId := 2,
    iOverride := 1000000,
    bExecute := FiFo_SetChannelOverride.bExecute,
    bErr => FiFo_Override_output.Error,
    iErrId => FiFo_Override_output.ErrorID); // FiFoSetChannelOverride
FiFo_Override_output.Busy := FiFo_SetChannelOverride.bBusy;

// NETWORK 10
FiFo_Start(
    iChannelId := 2,
    bExecute := start_do,
    bErr => fifo_startoutput.Error,
    iErrId => fifo_startoutput.ErrorID); // FiFoStart
fifo_startoutput.Busy := FiFo_Start.bBusy;

// NETWORK 11
FiFo_Stop(
    iChannelId := 2,
    bExecute := stop_do,
    bErr => fifo_stopoutput.Error,
    iErrId => fifo_stopoutput.ErrorID); // FiFoStop
fifo_stopoutput.Busy := FiFo_Stop.bBusy;

// NETWORK 12
FiFo_Write(
    iChannelId := 2,
    AdrDataArray := adr(pos_arr1),
    iColDim := 6,
    iRowsToWrite := 200,
    bExecute := FIFO_write_do,
    bErr => FIFO_write_output.Error,
    iErrId => FIFO_write_output.ErrorID); // FiFoWrite
FIFO_write_output.Busy := FiFo_Write.bBusy;

// NETWORK 13
FiFo_OverWrite(
    iChannelId := 2,
    AdrDataArray := adr(pos_arr1),
    iColDim := 6,
    iRowsToWrite := 200,
    bExecute := FIFO_overwrite_do,
    bErr => FIFO_write_output.Error,
    iErrId => FIFO_write_output.ErrorID); // FiFoOverwrite
FIFO_write_output.Busy := FiFo_OverWrite.bBusy;
END_ACTION

ACTION setpositionGen:
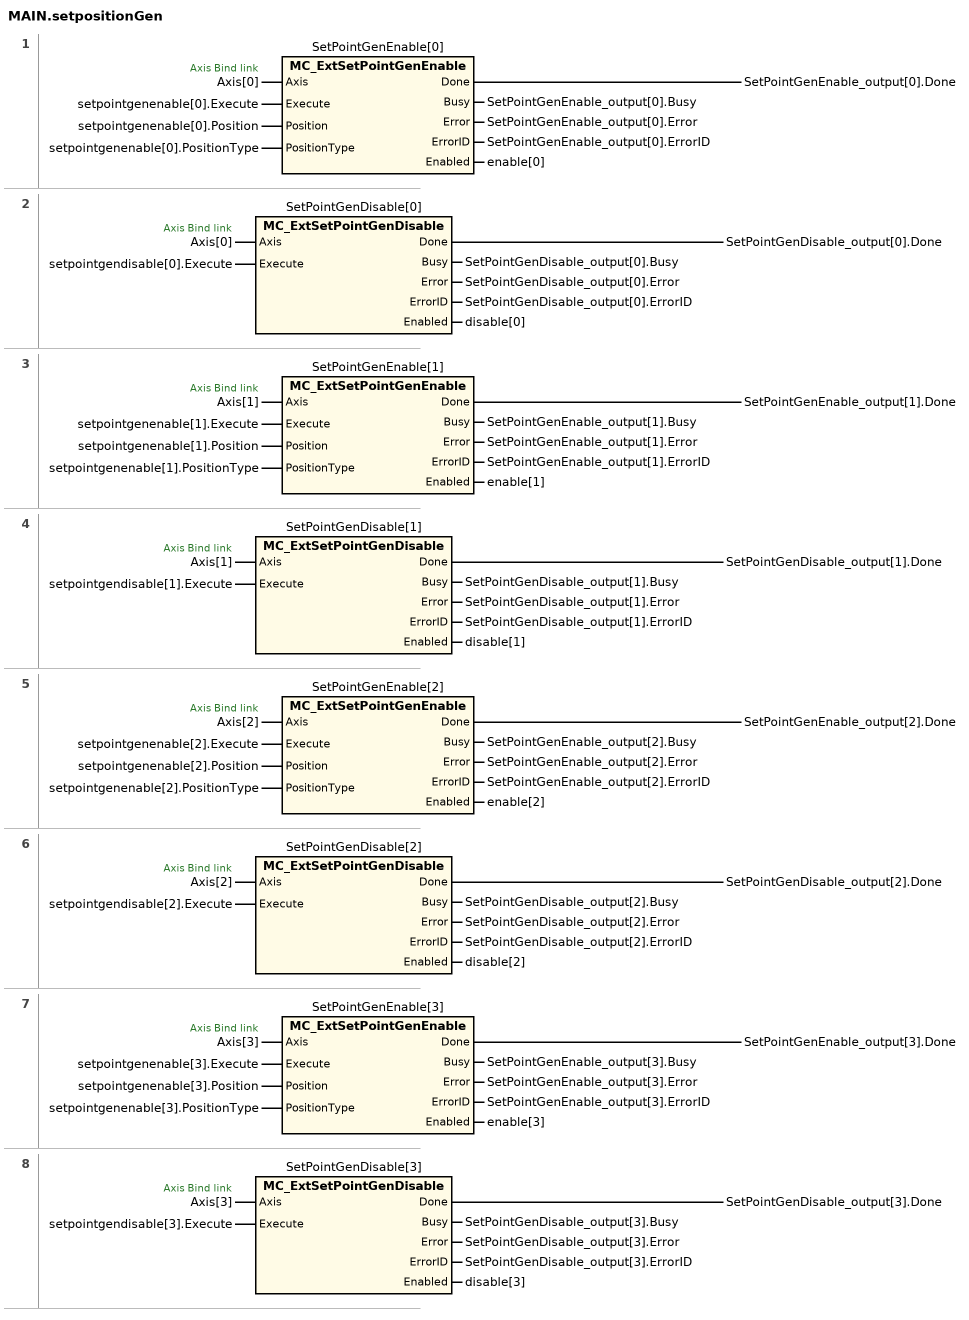
// NETWORK 1
//   Axis[0]: Axis Bind link
SetPointGenEnable[0](
    Axis := Axis[0],
    Execute := setpointgenenable[0].Execute,
    Position := setpointgenenable[0].Position,
    PositionType := setpointgenenable[0].PositionType,
    Busy => SetPointGenEnable_output[0].Busy,
    Error => SetPointGenEnable_output[0].Error,
    ErrorID => SetPointGenEnable_output[0].ErrorID,
    Enabled => enable[0]); // MC_ExtSetPointGenEnable
SetPointGenEnable_output[0].Done := SetPointGenEnable[0].Done;

// NETWORK 2
//   Axis[0]: Axis Bind link
SetPointGenDisable[0](
    Axis := Axis[0],
    Execute := setpointgendisable[0].Execute,
    Busy => SetPointGenDisable_output[0].Busy,
    Error => SetPointGenDisable_output[0].Error,
    ErrorID => SetPointGenDisable_output[0].ErrorID,
    Enabled => disable[0]); // MC_ExtSetPointGenDisable
SetPointGenDisable_output[0].Done := SetPointGenDisable[0].Done;

// NETWORK 3
//   Axis[1]: Axis Bind link
SetPointGenEnable[1](
    Axis := Axis[1],
    Execute := setpointgenenable[1].Execute,
    Position := setpointgenenable[1].Position,
    PositionType := setpointgenenable[1].PositionType,
    Busy => SetPointGenEnable_output[1].Busy,
    Error => SetPointGenEnable_output[1].Error,
    ErrorID => SetPointGenEnable_output[1].ErrorID,
    Enabled => enable[1]); // MC_ExtSetPointGenEnable
SetPointGenEnable_output[1].Done := SetPointGenEnable[1].Done;

// NETWORK 4
//   Axis[1]: Axis Bind link
SetPointGenDisable[1](
    Axis := Axis[1],
    Execute := setpointgendisable[1].Execute,
    Busy => SetPointGenDisable_output[1].Busy,
    Error => SetPointGenDisable_output[1].Error,
    ErrorID => SetPointGenDisable_output[1].ErrorID,
    Enabled => disable[1]); // MC_ExtSetPointGenDisable
SetPointGenDisable_output[1].Done := SetPointGenDisable[1].Done;

// NETWORK 5
//   Axis[2]: Axis Bind link
SetPointGenEnable[2](
    Axis := Axis[2],
    Execute := setpointgenenable[2].Execute,
    Position := setpointgenenable[2].Position,
    PositionType := setpointgenenable[2].PositionType,
    Busy => SetPointGenEnable_output[2].Busy,
    Error => SetPointGenEnable_output[2].Error,
    ErrorID => SetPointGenEnable_output[2].ErrorID,
    Enabled => enable[2]); // MC_ExtSetPointGenEnable
SetPointGenEnable_output[2].Done := SetPointGenEnable[2].Done;

// NETWORK 6
//   Axis[2]: Axis Bind link
SetPointGenDisable[2](
    Axis := Axis[2],
    Execute := setpointgendisable[2].Execute,
    Busy => SetPointGenDisable_output[2].Busy,
    Error => SetPointGenDisable_output[2].Error,
    ErrorID => SetPointGenDisable_output[2].ErrorID,
    Enabled => disable[2]); // MC_ExtSetPointGenDisable
SetPointGenDisable_output[2].Done := SetPointGenDisable[2].Done;

// NETWORK 7
//   Axis[3]: Axis Bind link
SetPointGenEnable[3](
    Axis := Axis[3],
    Execute := setpointgenenable[3].Execute,
    Position := setpointgenenable[3].Position,
    PositionType := setpointgenenable[3].PositionType,
    Busy => SetPointGenEnable_output[3].Busy,
    Error => SetPointGenEnable_output[3].Error,
    ErrorID => SetPointGenEnable_output[3].ErrorID,
    Enabled => enable[3]); // MC_ExtSetPointGenEnable
SetPointGenEnable_output[3].Done := SetPointGenEnable[3].Done;

// NETWORK 8
//   Axis[3]: Axis Bind link
SetPointGenDisable[3](
    Axis := Axis[3],
    Execute := setpointgendisable[3].Execute,
    Busy => SetPointGenDisable_output[3].Busy,
    Error => SetPointGenDisable_output[3].Error,
    ErrorID => SetPointGenDisable_output[3].ErrorID,
    Enabled => disable[3]); // MC_ExtSetPointGenDisable
SetPointGenDisable_output[3].Done := SetPointGenDisable[3].Done;

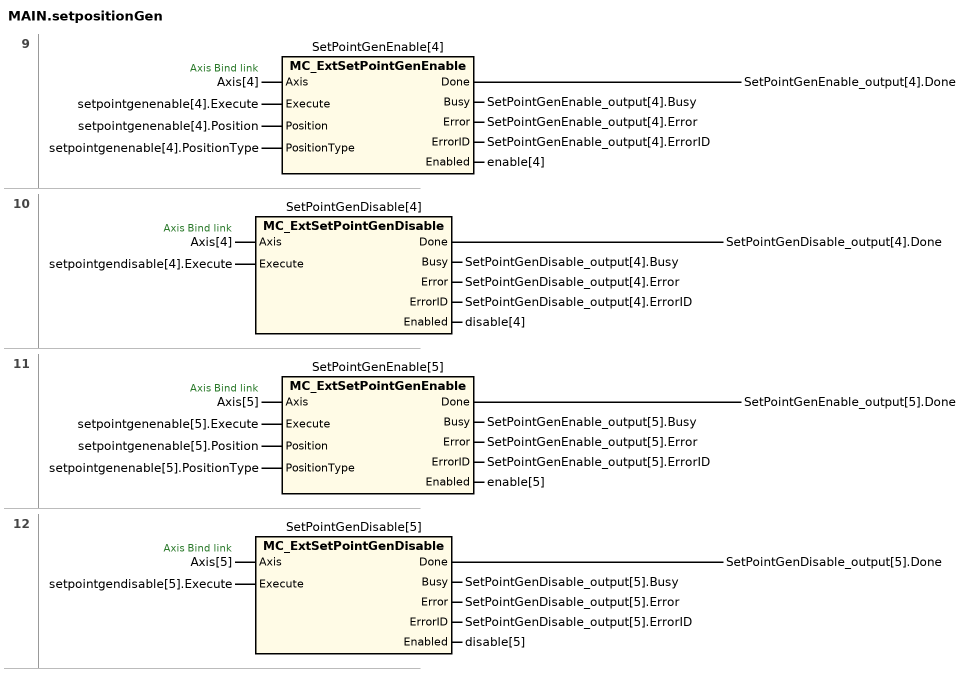
// NETWORK 9
//   Axis[4]: Axis Bind link
SetPointGenEnable[4](
    Axis := Axis[4],
    Execute := setpointgenenable[4].Execute,
    Position := setpointgenenable[4].Position,
    PositionType := setpointgenenable[4].PositionType,
    Busy => SetPointGenEnable_output[4].Busy,
    Error => SetPointGenEnable_output[4].Error,
    ErrorID => SetPointGenEnable_output[4].ErrorID,
    Enabled => enable[4]); // MC_ExtSetPointGenEnable
SetPointGenEnable_output[4].Done := SetPointGenEnable[4].Done;

// NETWORK 10
//   Axis[4]: Axis Bind link
SetPointGenDisable[4](
    Axis := Axis[4],
    Execute := setpointgendisable[4].Execute,
    Busy => SetPointGenDisable_output[4].Busy,
    Error => SetPointGenDisable_output[4].Error,
    ErrorID => SetPointGenDisable_output[4].ErrorID,
    Enabled => disable[4]); // MC_ExtSetPointGenDisable
SetPointGenDisable_output[4].Done := SetPointGenDisable[4].Done;

// NETWORK 11
//   Axis[5]: Axis Bind link
SetPointGenEnable[5](
    Axis := Axis[5],
    Execute := setpointgenenable[5].Execute,
    Position := setpointgenenable[5].Position,
    PositionType := setpointgenenable[5].PositionType,
    Busy => SetPointGenEnable_output[5].Busy,
    Error => SetPointGenEnable_output[5].Error,
    ErrorID => SetPointGenEnable_output[5].ErrorID,
    Enabled => enable[5]); // MC_ExtSetPointGenEnable
SetPointGenEnable_output[5].Done := SetPointGenEnable[5].Done;

// NETWORK 12
//   Axis[5]: Axis Bind link
SetPointGenDisable[5](
    Axis := Axis[5],
    Execute := setpointgendisable[5].Execute,
    Busy => SetPointGenDisable_output[5].Busy,
    Error => SetPointGenDisable_output[5].Error,
    ErrorID => SetPointGenDisable_output[5].ErrorID,
    Enabled => disable[5]); // MC_ExtSetPointGenDisable
SetPointGenDisable_output[5].Done := SetPointGenDisable[5].Done;
END_ACTION

END_PROGRAM

// ---- POUs/AxisStop.TcPOU
PROGRAM AxisStop
VAR	
	
END_VAR

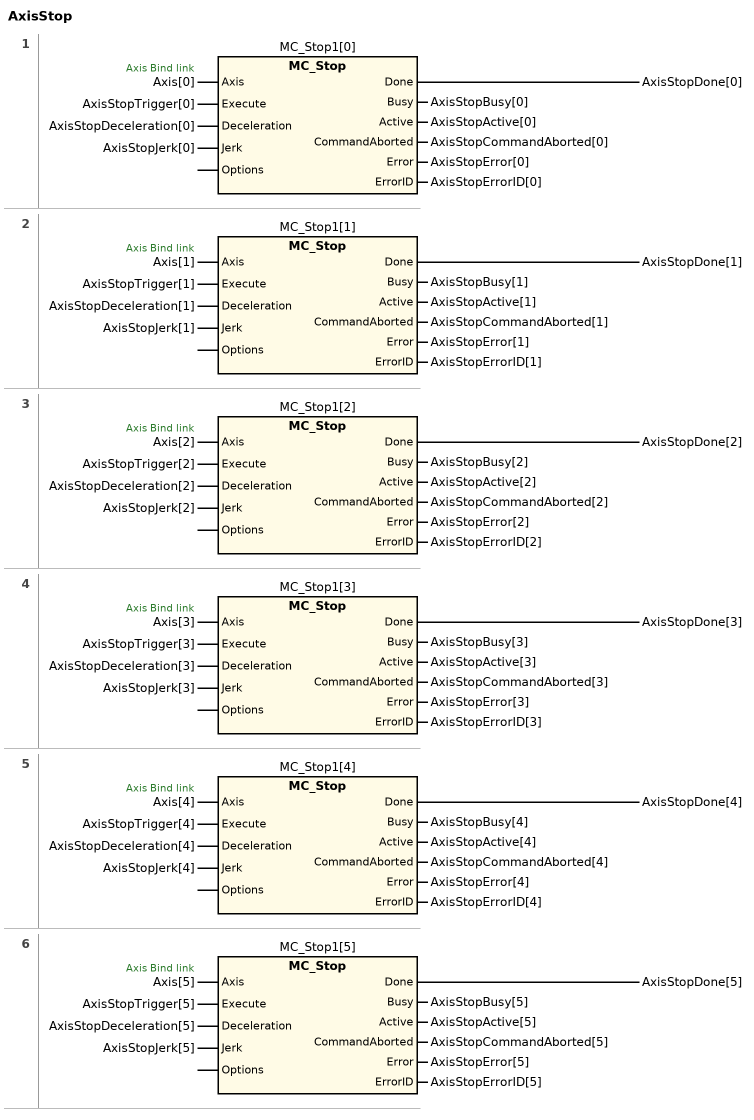
// NETWORK 1
//   MC_Stop1[0]: Axis Stop
//   Axis[0]: Axis Bind link
MC_Stop1[0](
    Axis := Axis[0],
    Execute := AxisStopTrigger[0],
    Deceleration := AxisStopDeceleration[0],
    Jerk := AxisStopJerk[0],
    Busy => AxisStopBusy[0],
    Active => AxisStopActive[0],
    CommandAborted => AxisStopCommandAborted[0],
    Error => AxisStopError[0],
    ErrorID => AxisStopErrorID[0]); // MC_Stop
AxisStopDone[0] := MC_Stop1[0].Done;

// NETWORK 2
//   MC_Stop1[1]: Axis Stop
//   Axis[1]: Axis Bind link
MC_Stop1[1](
    Axis := Axis[1],
    Execute := AxisStopTrigger[1],
    Deceleration := AxisStopDeceleration[1],
    Jerk := AxisStopJerk[1],
    Busy => AxisStopBusy[1],
    Active => AxisStopActive[1],
    CommandAborted => AxisStopCommandAborted[1],
    Error => AxisStopError[1],
    ErrorID => AxisStopErrorID[1]); // MC_Stop
AxisStopDone[1] := MC_Stop1[1].Done;

// NETWORK 3
//   MC_Stop1[2]: Axis Stop
//   Axis[2]: Axis Bind link
MC_Stop1[2](
    Axis := Axis[2],
    Execute := AxisStopTrigger[2],
    Deceleration := AxisStopDeceleration[2],
    Jerk := AxisStopJerk[2],
    Busy => AxisStopBusy[2],
    Active => AxisStopActive[2],
    CommandAborted => AxisStopCommandAborted[2],
    Error => AxisStopError[2],
    ErrorID => AxisStopErrorID[2]); // MC_Stop
AxisStopDone[2] := MC_Stop1[2].Done;

// NETWORK 4
//   MC_Stop1[3]: Axis Stop
//   Axis[3]: Axis Bind link
MC_Stop1[3](
    Axis := Axis[3],
    Execute := AxisStopTrigger[3],
    Deceleration := AxisStopDeceleration[3],
    Jerk := AxisStopJerk[3],
    Busy => AxisStopBusy[3],
    Active => AxisStopActive[3],
    CommandAborted => AxisStopCommandAborted[3],
    Error => AxisStopError[3],
    ErrorID => AxisStopErrorID[3]); // MC_Stop
AxisStopDone[3] := MC_Stop1[3].Done;

// NETWORK 5
//   MC_Stop1[4]: Axis Stop
//   Axis[4]: Axis Bind link
MC_Stop1[4](
    Axis := Axis[4],
    Execute := AxisStopTrigger[4],
    Deceleration := AxisStopDeceleration[4],
    Jerk := AxisStopJerk[4],
    Busy => AxisStopBusy[4],
    Active => AxisStopActive[4],
    CommandAborted => AxisStopCommandAborted[4],
    Error => AxisStopError[4],
    ErrorID => AxisStopErrorID[4]); // MC_Stop
AxisStopDone[4] := MC_Stop1[4].Done;

// NETWORK 6
//   MC_Stop1[5]: Axis Stop
//   Axis[5]: Axis Bind link
MC_Stop1[5](
    Axis := Axis[5],
    Execute := AxisStopTrigger[5],
    Deceleration := AxisStopDeceleration[5],
    Jerk := AxisStopJerk[5],
    Busy => AxisStopBusy[5],
    Active => AxisStopActive[5],
    CommandAborted => AxisStopCommandAborted[5],
    Error => AxisStopError[5],
    ErrorID => AxisStopErrorID[5]); // MC_Stop
AxisStopDone[5] := MC_Stop1[5].Done;

END_PROGRAM

// ---- POUs/Move_JOG.TcPOU
PROGRAM Move_JOG
VAR
	
END_VAR

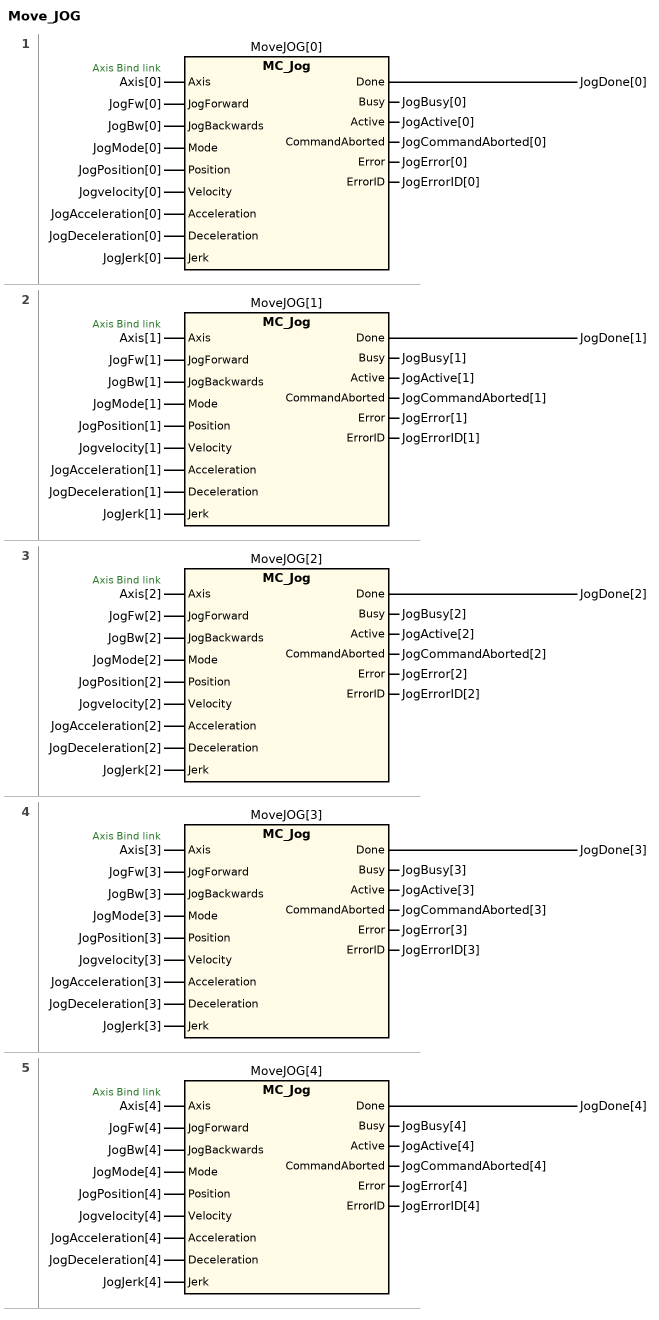
// NETWORK 1
//   MoveJOG[0]: MoveJOG
//   Axis[0]: Axis Bind link
MoveJOG[0](
    Axis := Axis[0],
    JogForward := JogFw[0],
    JogBackwards := JogBw[0],
    Mode := JogMode[0],
    Position := JogPosition[0],
    Velocity := Jogvelocity[0],
    Acceleration := JogAcceleration[0],
    Deceleration := JogDeceleration[0],
    Jerk := JogJerk[0],
    Busy => JogBusy[0],
    Active => JogActive[0],
    CommandAborted => JogCommandAborted[0],
    Error => JogError[0],
    ErrorID => JogErrorID[0]); // MC_Jog
JogDone[0] := MoveJOG[0].Done;

// NETWORK 2
//   MoveJOG[1]: MoveJOG
//   Axis[1]: Axis Bind link
MoveJOG[1](
    Axis := Axis[1],
    JogForward := JogFw[1],
    JogBackwards := JogBw[1],
    Mode := JogMode[1],
    Position := JogPosition[1],
    Velocity := Jogvelocity[1],
    Acceleration := JogAcceleration[1],
    Deceleration := JogDeceleration[1],
    Jerk := JogJerk[1],
    Busy => JogBusy[1],
    Active => JogActive[1],
    CommandAborted => JogCommandAborted[1],
    Error => JogError[1],
    ErrorID => JogErrorID[1]); // MC_Jog
JogDone[1] := MoveJOG[1].Done;

// NETWORK 3
//   MoveJOG[2]: MoveJOG
//   Axis[2]: Axis Bind link
MoveJOG[2](
    Axis := Axis[2],
    JogForward := JogFw[2],
    JogBackwards := JogBw[2],
    Mode := JogMode[2],
    Position := JogPosition[2],
    Velocity := Jogvelocity[2],
    Acceleration := JogAcceleration[2],
    Deceleration := JogDeceleration[2],
    Jerk := JogJerk[2],
    Busy => JogBusy[2],
    Active => JogActive[2],
    CommandAborted => JogCommandAborted[2],
    Error => JogError[2],
    ErrorID => JogErrorID[2]); // MC_Jog
JogDone[2] := MoveJOG[2].Done;

// NETWORK 4
//   MoveJOG[3]: MoveJOG
//   Axis[3]: Axis Bind link
MoveJOG[3](
    Axis := Axis[3],
    JogForward := JogFw[3],
    JogBackwards := JogBw[3],
    Mode := JogMode[3],
    Position := JogPosition[3],
    Velocity := Jogvelocity[3],
    Acceleration := JogAcceleration[3],
    Deceleration := JogDeceleration[3],
    Jerk := JogJerk[3],
    Busy => JogBusy[3],
    Active => JogActive[3],
    CommandAborted => JogCommandAborted[3],
    Error => JogError[3],
    ErrorID => JogErrorID[3]); // MC_Jog
JogDone[3] := MoveJOG[3].Done;

// NETWORK 5
//   MoveJOG[4]: MoveJOG
//   Axis[4]: Axis Bind link
MoveJOG[4](
    Axis := Axis[4],
    JogForward := JogFw[4],
    JogBackwards := JogBw[4],
    Mode := JogMode[4],
    Position := JogPosition[4],
    Velocity := Jogvelocity[4],
    Acceleration := JogAcceleration[4],
    Deceleration := JogDeceleration[4],
    Jerk := JogJerk[4],
    Busy => JogBusy[4],
    Active => JogActive[4],
    CommandAborted => JogCommandAborted[4],
    Error => JogError[4],
    ErrorID => JogErrorID[4]); // MC_Jog
JogDone[4] := MoveJOG[4].Done;

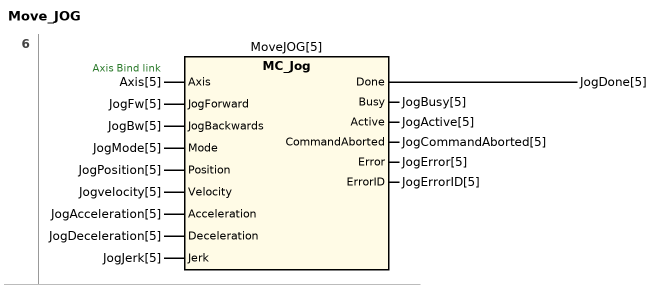
// NETWORK 6
//   MoveJOG[5]: MoveJOG
//   Axis[5]: Axis Bind link
MoveJOG[5](
    Axis := Axis[5],
    JogForward := JogFw[5],
    JogBackwards := JogBw[5],
    Mode := JogMode[5],
    Position := JogPosition[5],
    Velocity := Jogvelocity[5],
    Acceleration := JogAcceleration[5],
    Deceleration := JogDeceleration[5],
    Jerk := JogJerk[5],
    Busy => JogBusy[5],
    Active => JogActive[5],
    CommandAborted => JogCommandAborted[5],
    Error => JogError[5],
    ErrorID => JogErrorID[5]); // MC_Jog
JogDone[5] := MoveJOG[5].Done;

END_PROGRAM

// ---- POUs/AxisMoveAbsoulte.TcPOU
PROGRAM AxisMoveAbsoulte
VAR
END_VAR

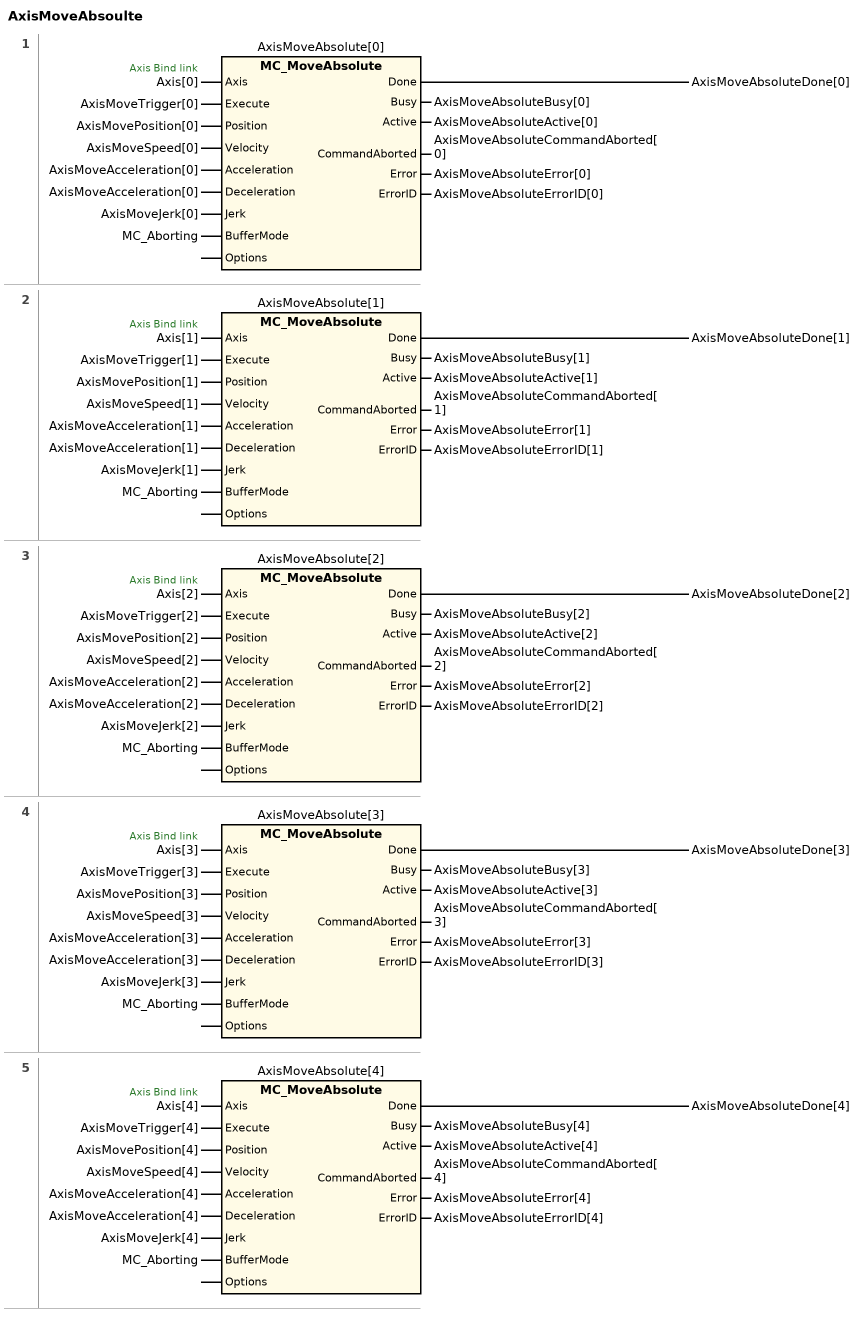
// NETWORK 1
//   AxisMoveAbsolute[0]: Axis Move Absolute
//   Axis[0]: Axis Bind link
AxisMoveAbsolute[0](
    Axis := Axis[0],
    Execute := AxisMoveTrigger[0],
    Position := AxisMovePosition[0],
    Velocity := AxisMoveSpeed[0],
    Acceleration := AxisMoveAcceleration[0],
    Deceleration := AxisMoveAcceleration[0],
    Jerk := AxisMoveJerk[0],
    BufferMode := MC_Aborting,
    Busy => AxisMoveAbsoluteBusy[0],
    Active => AxisMoveAbsoluteActive[0],
    CommandAborted => AxisMoveAbsoluteCommandAborted[0],
    Error => AxisMoveAbsoluteError[0],
    ErrorID => AxisMoveAbsoluteErrorID[0]); // MC_MoveAbsolute
AxisMoveAbsoluteDone[0] := AxisMoveAbsolute[0].Done;

// NETWORK 2
//   AxisMoveAbsolute[1]: Axis Move Absolute
//   Axis[1]: Axis Bind link
AxisMoveAbsolute[1](
    Axis := Axis[1],
    Execute := AxisMoveTrigger[1],
    Position := AxisMovePosition[1],
    Velocity := AxisMoveSpeed[1],
    Acceleration := AxisMoveAcceleration[1],
    Deceleration := AxisMoveAcceleration[1],
    Jerk := AxisMoveJerk[1],
    BufferMode := MC_Aborting,
    Busy => AxisMoveAbsoluteBusy[1],
    Active => AxisMoveAbsoluteActive[1],
    CommandAborted => AxisMoveAbsoluteCommandAborted[1],
    Error => AxisMoveAbsoluteError[1],
    ErrorID => AxisMoveAbsoluteErrorID[1]); // MC_MoveAbsolute
AxisMoveAbsoluteDone[1] := AxisMoveAbsolute[1].Done;

// NETWORK 3
//   AxisMoveAbsolute[2]: Axis Move Absolute
//   Axis[2]: Axis Bind link
AxisMoveAbsolute[2](
    Axis := Axis[2],
    Execute := AxisMoveTrigger[2],
    Position := AxisMovePosition[2],
    Velocity := AxisMoveSpeed[2],
    Acceleration := AxisMoveAcceleration[2],
    Deceleration := AxisMoveAcceleration[2],
    Jerk := AxisMoveJerk[2],
    BufferMode := MC_Aborting,
    Busy => AxisMoveAbsoluteBusy[2],
    Active => AxisMoveAbsoluteActive[2],
    CommandAborted => AxisMoveAbsoluteCommandAborted[2],
    Error => AxisMoveAbsoluteError[2],
    ErrorID => AxisMoveAbsoluteErrorID[2]); // MC_MoveAbsolute
AxisMoveAbsoluteDone[2] := AxisMoveAbsolute[2].Done;

// NETWORK 4
//   AxisMoveAbsolute[3]: Axis Move Absolute
//   Axis[3]: Axis Bind link
AxisMoveAbsolute[3](
    Axis := Axis[3],
    Execute := AxisMoveTrigger[3],
    Position := AxisMovePosition[3],
    Velocity := AxisMoveSpeed[3],
    Acceleration := AxisMoveAcceleration[3],
    Deceleration := AxisMoveAcceleration[3],
    Jerk := AxisMoveJerk[3],
    BufferMode := MC_Aborting,
    Busy => AxisMoveAbsoluteBusy[3],
    Active => AxisMoveAbsoluteActive[3],
    CommandAborted => AxisMoveAbsoluteCommandAborted[3],
    Error => AxisMoveAbsoluteError[3],
    ErrorID => AxisMoveAbsoluteErrorID[3]); // MC_MoveAbsolute
AxisMoveAbsoluteDone[3] := AxisMoveAbsolute[3].Done;

// NETWORK 5
//   AxisMoveAbsolute[4]: Axis Move Absolute
//   Axis[4]: Axis Bind link
AxisMoveAbsolute[4](
    Axis := Axis[4],
    Execute := AxisMoveTrigger[4],
    Position := AxisMovePosition[4],
    Velocity := AxisMoveSpeed[4],
    Acceleration := AxisMoveAcceleration[4],
    Deceleration := AxisMoveAcceleration[4],
    Jerk := AxisMoveJerk[4],
    BufferMode := MC_Aborting,
    Busy => AxisMoveAbsoluteBusy[4],
    Active => AxisMoveAbsoluteActive[4],
    CommandAborted => AxisMoveAbsoluteCommandAborted[4],
    Error => AxisMoveAbsoluteError[4],
    ErrorID => AxisMoveAbsoluteErrorID[4]); // MC_MoveAbsolute
AxisMoveAbsoluteDone[4] := AxisMoveAbsolute[4].Done;

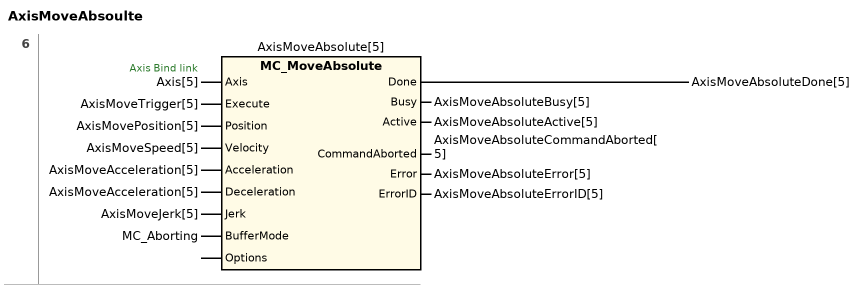
// NETWORK 6
//   AxisMoveAbsolute[5]: Axis Move Absolute
//   Axis[5]: Axis Bind link
AxisMoveAbsolute[5](
    Axis := Axis[5],
    Execute := AxisMoveTrigger[5],
    Position := AxisMovePosition[5],
    Velocity := AxisMoveSpeed[5],
    Acceleration := AxisMoveAcceleration[5],
    Deceleration := AxisMoveAcceleration[5],
    Jerk := AxisMoveJerk[5],
    BufferMode := MC_Aborting,
    Busy => AxisMoveAbsoluteBusy[5],
    Active => AxisMoveAbsoluteActive[5],
    CommandAborted => AxisMoveAbsoluteCommandAborted[5],
    Error => AxisMoveAbsoluteError[5],
    ErrorID => AxisMoveAbsoluteErrorID[5]); // MC_MoveAbsolute
AxisMoveAbsoluteDone[5] := AxisMoveAbsolute[5].Done;

END_PROGRAM

// ---- POUs/Homing.TcPOU
PROGRAM Homing
VAR
	
END_VAR

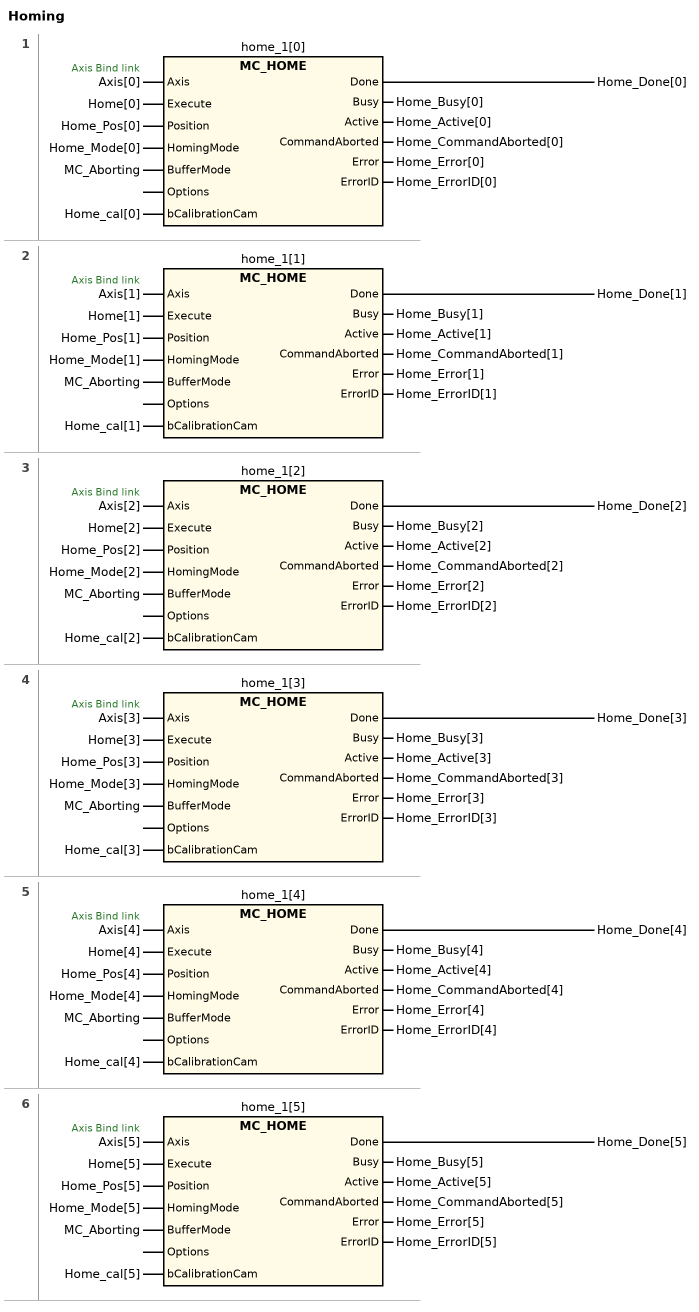
// NETWORK 1
//   home_1[0]: HOME
//   Axis[0]: Axis Bind link
home_1[0](
    Axis := Axis[0],
    Execute := Home[0],
    Position := Home_Pos[0],
    HomingMode := Home_Mode[0],
    BufferMode := MC_Aborting,
    bCalibrationCam := Home_cal[0],
    Busy => Home_Busy[0],
    Active => Home_Active[0],
    CommandAborted => Home_CommandAborted[0],
    Error => Home_Error[0],
    ErrorID => Home_ErrorID[0]); // MC_HOME
Home_Done[0] := home_1[0].Done;

// NETWORK 2
//   home_1[1]: HOME
//   Axis[1]: Axis Bind link
home_1[1](
    Axis := Axis[1],
    Execute := Home[1],
    Position := Home_Pos[1],
    HomingMode := Home_Mode[1],
    BufferMode := MC_Aborting,
    bCalibrationCam := Home_cal[1],
    Busy => Home_Busy[1],
    Active => Home_Active[1],
    CommandAborted => Home_CommandAborted[1],
    Error => Home_Error[1],
    ErrorID => Home_ErrorID[1]); // MC_HOME
Home_Done[1] := home_1[1].Done;

// NETWORK 3
//   home_1[2]: HOME
//   Axis[2]: Axis Bind link
home_1[2](
    Axis := Axis[2],
    Execute := Home[2],
    Position := Home_Pos[2],
    HomingMode := Home_Mode[2],
    BufferMode := MC_Aborting,
    bCalibrationCam := Home_cal[2],
    Busy => Home_Busy[2],
    Active => Home_Active[2],
    CommandAborted => Home_CommandAborted[2],
    Error => Home_Error[2],
    ErrorID => Home_ErrorID[2]); // MC_HOME
Home_Done[2] := home_1[2].Done;

// NETWORK 4
//   home_1[3]: HOME
//   Axis[3]: Axis Bind link
home_1[3](
    Axis := Axis[3],
    Execute := Home[3],
    Position := Home_Pos[3],
    HomingMode := Home_Mode[3],
    BufferMode := MC_Aborting,
    bCalibrationCam := Home_cal[3],
    Busy => Home_Busy[3],
    Active => Home_Active[3],
    CommandAborted => Home_CommandAborted[3],
    Error => Home_Error[3],
    ErrorID => Home_ErrorID[3]); // MC_HOME
Home_Done[3] := home_1[3].Done;

// NETWORK 5
//   home_1[4]: HOME
//   Axis[4]: Axis Bind link
home_1[4](
    Axis := Axis[4],
    Execute := Home[4],
    Position := Home_Pos[4],
    HomingMode := Home_Mode[4],
    BufferMode := MC_Aborting,
    bCalibrationCam := Home_cal[4],
    Busy => Home_Busy[4],
    Active => Home_Active[4],
    CommandAborted => Home_CommandAborted[4],
    Error => Home_Error[4],
    ErrorID => Home_ErrorID[4]); // MC_HOME
Home_Done[4] := home_1[4].Done;

// NETWORK 6
//   home_1[5]: HOME
//   Axis[5]: Axis Bind link
home_1[5](
    Axis := Axis[5],
    Execute := Home[5],
    Position := Home_Pos[5],
    HomingMode := Home_Mode[5],
    BufferMode := MC_Aborting,
    bCalibrationCam := Home_cal[5],
    Busy => Home_Busy[5],
    Active => Home_Active[5],
    CommandAborted => Home_CommandAborted[5],
    Error => Home_Error[5],
    ErrorID => Home_ErrorID[5]); // MC_HOME
Home_Done[5] := home_1[5].Done;

END_PROGRAM

// ---- POUs/AxisReset.TcPOU
PROGRAM AxisReset
VAR

END_VAR

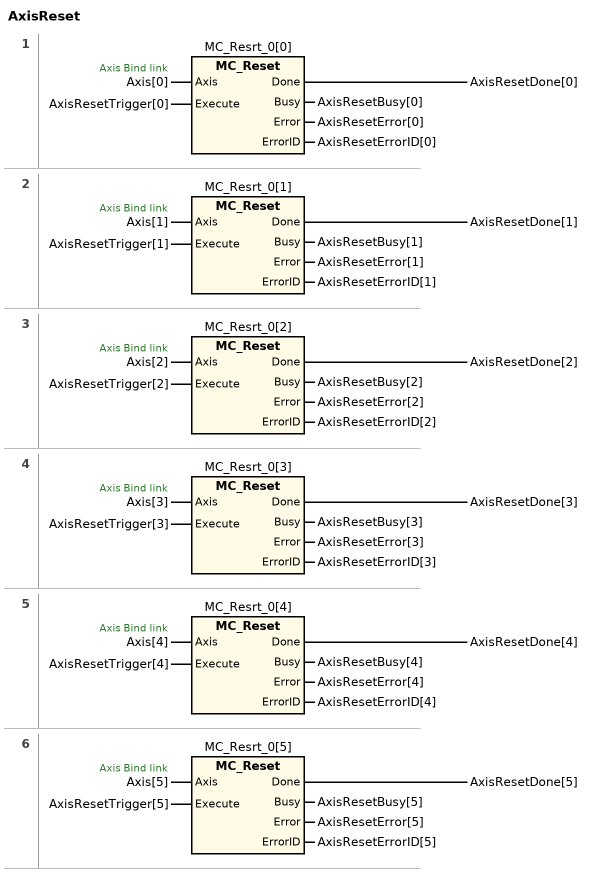
// NETWORK 1
//   MC_Resrt_0[0]: Reset
//   Axis[0]: Axis Bind link
MC_Resrt_0[0](
    Axis := Axis[0],
    Execute := AxisResetTrigger[0],
    Busy => AxisResetBusy[0],
    Error => AxisResetError[0],
    ErrorID => AxisResetErrorID[0]); // MC_Reset
AxisResetDone[0] := MC_Resrt_0[0].Done;

// NETWORK 2
//   MC_Resrt_0[1]: Reset
//   Axis[1]: Axis Bind link
MC_Resrt_0[1](
    Axis := Axis[1],
    Execute := AxisResetTrigger[1],
    Busy => AxisResetBusy[1],
    Error => AxisResetError[1],
    ErrorID => AxisResetErrorID[1]); // MC_Reset
AxisResetDone[1] := MC_Resrt_0[1].Done;

// NETWORK 3
//   MC_Resrt_0[2]: Reset
//   Axis[2]: Axis Bind link
MC_Resrt_0[2](
    Axis := Axis[2],
    Execute := AxisResetTrigger[2],
    Busy => AxisResetBusy[2],
    Error => AxisResetError[2],
    ErrorID => AxisResetErrorID[2]); // MC_Reset
AxisResetDone[2] := MC_Resrt_0[2].Done;

// NETWORK 4
//   MC_Resrt_0[3]: Reset
//   Axis[3]: Axis Bind link
MC_Resrt_0[3](
    Axis := Axis[3],
    Execute := AxisResetTrigger[3],
    Busy => AxisResetBusy[3],
    Error => AxisResetError[3],
    ErrorID => AxisResetErrorID[3]); // MC_Reset
AxisResetDone[3] := MC_Resrt_0[3].Done;

// NETWORK 5
//   MC_Resrt_0[4]: Reset
//   Axis[4]: Axis Bind link
MC_Resrt_0[4](
    Axis := Axis[4],
    Execute := AxisResetTrigger[4],
    Busy => AxisResetBusy[4],
    Error => AxisResetError[4],
    ErrorID => AxisResetErrorID[4]); // MC_Reset
AxisResetDone[4] := MC_Resrt_0[4].Done;

// NETWORK 6
//   MC_Resrt_0[5]: Reset
//   Axis[5]: Axis Bind link
MC_Resrt_0[5](
    Axis := Axis[5],
    Execute := AxisResetTrigger[5],
    Busy => AxisResetBusy[5],
    Error => AxisResetError[5],
    ErrorID => AxisResetErrorID[5]); // MC_Reset
AxisResetDone[5] := MC_Resrt_0[5].Done;

END_PROGRAM

// ---- POUs/CSV read_write in text mode/P_TextModeWrite.TcPOU
(* Writing of CSV file in text mode. None of the field value is containing any non-printing control characters like line feed, carriage return, quotation marks, semicolon... *)
PROGRAM P_TextModeWrite
VAR
	bWrite			: BOOL := FALSE;(* Rising edge starts program execution *)
	sNetId			: T_AmsNetId := '';	(* TwinCAT system network address *)
	sFileName		: T_MaxString := 'C:\Temp\TextModeGen.csv';(* CSV destination file path and name *)
	sCSVLine		: T_MaxString := '';(* Single CSV text line (row, record), we are using string as record buffer (your are able to see created fields) *)
	sCSVField		: T_MaxString := '';(* Single CSV field value (column, record field) *)
	bBusy			: BOOL;
	bError			: BOOL;
	nErrId			: UDINT;
	nRow	 		: UDINT 	:= 0;(* Row number (record) *)
	nColumn			: UDINT 	:= 0;(* Column number (record field) *)
	hFile			: UINT		:= 0;(* File handle of the source file *)
	step			: DWORD 	:= 0;
	fbFileOpen		: FB_FileOpen;(* Opens file *)
	fbFileClose		: FB_FileClose;(* Closes file *)
	fbFilePuts		: FB_FilePuts;(* Writes one record (line) *)
	fbWriter		: FB_CSVMemBufferWriter;(* Helper function block used to create CSV data bytes (single record line) *)

	database		: ARRAY[0..MAX_CSV_ROWS, 0..MAX_CSV_COLUMNS ] OF STRING(MAX_CSV_FIELD_LENGTH) :=[ ];(* Source PLC database *)

END_VAR

bWrite:=MAIN.P_TextModeWrite_WriteTrigger;
sFileName:=MAIN.P_TextModeWrite_WriteFilePath;

CASE step OF
	0:	(* Wait for rising edge at bWrite variable *)
		IF bWrite THEN
			bWrite 	:= FALSE;
			bBusy 	:= TRUE;
			bError	:= FALSE;
			nErrId	:= 0;
			hFile	:= 0;
			nRow	:= 0;
			nColumn	:= 0;
			step 	:= 1;
		END_IF

	1:	(* Open source file *)
		fbFileOpen(  bExecute := FALSE  );
		fbFileOpen( sNetId := sNetId, sPathName := sFileName, nMode := FOPEN_MODEWRITE OR FOPEN_MODETEXT,(* Open file in TEXT mode! *)
					ePath := PATH_GENERIC, bExecute := TRUE );
		step := 2;

	2:(* Wait until open not busy *)
		fbFileOpen( bExecute := FALSE, bError => bError, nErrID => nErrID, hFile => hFile );
		IF NOT fbFileOpen.bBusy THEN
			IF NOT fbFileOpen.bError THEN
				step := 3;
			ELSE(* Error: file not found? *)
				step := 100;
			END_IF
		END_IF

	3:(* Convert one PLC record to CSV format *)
		sCSVLine := '';
		fbWriter.eCmd := eEnumCmd_First;(* Write first field value *)
		IF nRow <= MAX_CSV_ROWS THEN

			FOR nColumn := 0 TO MAX_CSV_COLUMNS BY 1 DO

				sCSVField := STRING_TO_CSVFIELD( database[ nRow, nColumn ], FALSE );(* TODO: Get field value from your application *)

				(* Add new field to the record buffer *)
				fbWriter( 	pBuffer := ADR( sCSVLine ), cbBuffer := SIZEOF( sCSVLine ) - 1, putValue := sCSVField, pValue := 0, cbValue := 0,
							bCRLF := ( nColumn = MAX_CSV_COLUMNS ) );(* bCRLF == TRUE => Write CRLF after the last field value *)
				IF fbWriter.bOk THEN
					fbWriter.eCmd := eEnumCmd_Next;(* Write next field value *)
				ELSE(* Error *)
					step := 100;
					RETURN;
				END_IF

			END_FOR(* FOR nColumn := 0... *)

			(* FB_FilePuts adds allready CR (carriage return) to the written line.
			We have to replace the $R$L characters with $L character to avoid double CR. *)
			IF RIGHT( sCSVLine, 2 ) = '$R$L' THEN
				sCSVLine := REPLACE( sCSVLine, '$L', 2, LEN( sCSVLine ) - 1 );
			END_IF

			nRow := nRow + 1;(* Increment number of created records (rows) *)
			step := 4;(* Write record to the file *)

		ELSE(* All rows written => Close file *)
			step := 10;
		END_IF

	4:	(* Write single text line *)
		fbFilePuts( bExecute := FALSE );
		fbFilePuts( sNetId := sNetId, hFile := hFile, sLine := sCSVLine, bExecute := TRUE );
		step := 5;

	5:(* Wait until write not busy *)
		fbFilePuts( bExecute := FALSE, bError => bError, nErrID => nErrID );
		IF NOT fbFilePuts.bBusy THEN
			IF NOT fbFilePuts.bError THEN
				step := 3;(* Write next record *)
			ELSE(* Error *)
				step := 100;
			END_IF
		END_IF

	10:	(* Close source file *)
		fbFileClose( bExecute := FALSE );
		fbFileClose( sNetId := sNetId, hFile := hFile, bExecute := TRUE );
		step := 11;

	11:(* Wait until close not busy *)
		fbFileClose( bExecute := FALSE, bError => bError, nErrID => nErrID );
		IF ( NOT fbFileClose.bBusy ) THEN
			hFile := 0;
			step := 100;
		END_IF

	100: (* Error or ready step => cleanup *)
		IF ( hFile <> 0 ) THEN
			step := 10; (* Close the source file *)
		ELSE
			bBusy := FALSE;
			step := 0;	(* Ready *)
		END_IF

END_CASE

END_PROGRAM

// ---- POUs/CSV read_write in text mode/P_TextModeRead.TcPOU
(* Reading of CSV file in text mode. None of the field value is containing any non-printing control characters like line feed, carriage return, quotation marks, semicolon... *)
PROGRAM P_TextModeRead
VAR
	bRead			: BOOL := FALSE;(* Rising edge starts program execution *)
	sNetId			: T_AmsNetId := '';	(* TwinCAT system network address *)
	sFileName		: T_MaxString := 'C:\Temp\TextModeGen.csv';(* CSV source file path and name *)
	sCSVLine		: T_MaxString := '';(* Single CSV text line (row, record), we are using string as record buffer (your are able to see read fields)  *)
	sCSVField		: T_MaxString := '';(* Single CSV field value (column, record field) *)
	bBusy			: BOOL;
	bError			: BOOL;
	nErrId			: UDINT;
	nRow	 		: UDINT 	:= 0;(* Row number (record) *)
	nColumn			: UDINT 	:= 0;(* Column number (record field) *)
	hFile			: UINT		:= 0;(* File handle of the source file *)
	step			: DWORD 	:= 0;
	fbFileOpen		: FB_FileOpen;(* Opens file *)
	fbFileClose		: FB_FileClose;(* Closes file *)
	fbFileGets		: FB_FileGets;(* Reads one record (line) *)
	fbReader		: FB_CSVMemBufferReader;(* Helper function block used to parse CSV data bytes (single record line) *)

	database		: ARRAY[0..MAX_CSV_ROWS, 0..MAX_CSV_COLUMNS ] OF STRING(MAX_CSV_FIELD_LENGTH);(* Target PLC database *)
END_VAR

bRead:=MAIN.P_TextModeRead_ReadTrigger;
sFileName:=MAIN.P_TextModeRead_ReadFilePath;


CASE step OF
	0:	(* Wait for rising edge at bRead variable *)
		IF bRead THEN
			bRead 	:= FALSE;
			bBusy 	:= TRUE;
			bError	:= FALSE;
			nErrId	:= 0;
			hFile	:= 0;
			nRow	:= 0;
			nColumn	:= 0;
			MEMSET( ADR( database ), 0, SIZEOF( database ) );
			step 		:= 1;
		END_IF

	1:	(* Open source file *)
		fbFileOpen(  bExecute := FALSE  );
		fbFileOpen( sNetId := sNetId, sPathName := sFileName, nMode := FOPEN_MODEREAD OR FOPEN_MODETEXT,(* Open file in TEXT mode! *)
					ePath := PATH_GENERIC, bExecute := TRUE );
		step := 2;

	2:(* Wait until open not busy *)
		fbFileOpen( bExecute := FALSE, bError => bError, nErrID => nErrID, hFile => hFile );
		IF NOT fbFileOpen.bBusy THEN
			IF NOT fbFileOpen.bError THEN
				step := 3;
			ELSE(* Error: file not found? *)
				step := 100;
			END_IF
		END_IF

	3:	(* Read single line (record) *)
		fbFileGets( bExecute := FALSE );
		fbFileGets( sNetId := sNetId, hFile := hFile, bExecute := TRUE );
		step := 4;

	4:(* Wait until read not busy *)
		fbFileGets( bExecute := FALSE, bError => bError, nErrID => nErrID, sLine => sCSVLine );
		IF NOT fbFileGets.bBusy THEN
			IF NOT fbFileGets.bError THEN
				IF fbFileGets.bEOF THEN
					step := 10;(* End of file reached => Close source file *)
				ELSE

					(* FB_FileGets returns text line without the CR (carriage return) character.
					We have to restore the CR character (replace the $L character with $R$L characters) *)
					IF RIGHT( sCSVLine, 1 ) = '$L' THEN
						sCSVLine := REPLACE( sCSVLine, '$R$L', 2, LEN( sCSVLine ) );
					END_IF

					step := 5;
				END_IF
			ELSE(* Error *)
				step := 100;
			END_IF
		END_IF

	5:(* Parse single line (record) *)
		fbReader.eCmd := eEnumCmd_First;(* Read first field value *)
		REPEAT
			fbReader( pBuffer := ADR( sCSVLine ), cbBuffer := SIZEOF( sCSVLine ), getValue => sCSVField );
			IF fbReader.bOk THEN
				fbReader.eCmd := eEnumCmd_Next;(* Read next field value *)

				IF ( nRow <= MAX_CSV_ROWS ) THEN
					IF ( nColumn <= MAX_CSV_COLUMNS ) THEN
						database[nRow, nColumn] := CSVFIELD_TO_STRING( sCSVField, FALSE );(* TODO: Save or use the field value in your application *)
					END_IF
				END_IF

				nColumn := nColumn + 1;(* Increment number of read columns *)
				IF fbReader.bCRLF THEN(* CRLF == TRUE => End of reacord reached *)
					nRow 		:= nRow + 1;(* Increment number of read records *)
					nColumn 	:= 0;(* Reset number of columns *)
				END_IF

			ELSE(* Error: End of record reached or all fields read *)
				step := 3;(* Try to read next line *)
			END_IF
		UNTIL NOT fbReader.bOk
		END_REPEAT

	10:	(* Close source file *)
		fbFileClose( bExecute := FALSE );
		fbFileClose( sNetId := sNetId, hFile := hFile, bExecute := TRUE );
		step := 11;

	11:(* Wait until close not busy *)
		fbFileClose( bExecute := FALSE, bError => bError, nErrID => nErrID );
		IF ( NOT fbFileClose.bBusy ) THEN
			hFile := 0;
			step := 100;
		END_IF

	100: (* Error or ready step => cleanup *)
		IF ( hFile <> 0 ) THEN
			step := 10; (* Close the source file *)
		ELSE
			bBusy := FALSE;
			step := 0;	(* Ready *)
		END_IF

END_CASE

END_PROGRAM

// ---- GlobalTextList.TcGTLO
TEXTLIST GlobalTextList
  10 = '%.3f'
  8 = '%d'
  30 = '%f'
  6 = '%s'
  38 = '+'
  40 = '++'
  37 = '-'
  39 = '--'
  26 = 'Actual Position:'
  27 = 'Actual Speed:'
  25 = 'ActualPosition:'
  9 = 'Axis State'
  23 = 'Axis1'
  55 = 'A点'
  114 = 'ChannelOv'
  113 = 'ChannelOver'
  116 = 'ChOverride'
  21 = 'Current Job State'
  22 = 'Current Job State:'
  7 = 'Current Job State：'
  20 = 'Current Job:'
  5 = 'Current Job：'
  14 = 'Current Position:'
  15 = 'Current Speed:'
  11 = 'CurrentJobState'
  18 = 'CurrentJobState:'
  119 = 'DisGroup'
  34 = 'DOWN'
  102 = 'FIFO:%d'
  104 = 'FIFO_'
  110 = 'FIFO_)top'
  108 = 'FIFO_Disin'
  107 = 'FIFO_in'
  115 = 'FIFO_inte'
  106 = 'FIFO_overwrite'
  111 = 'FIFO_S'
  109 = 'FIFO_start'
  112 = 'FIFO_Stop'
  103 = 'FIFO_write'
  101 = 'FIFO长度:%d'
  0 = 'Global State'
  120 = 'Group'
  52 = 'HOME'
  3 = 'Init'
  118 = 'Integrate'
  17 = 'ModeOfOperation:'
  4 = 'MOVE'
  33 = 'MOVE DOWN'
  32 = 'MOVE UP'
  31 = 'moveup'
  2 = 'OFF'
  1 = 'ON'
  28 = 'Operation Mode'
  29 = 'Operation Mode:'
  122 = 'Override'
  105 = 'overwrite'
  117 = 'Overwrite'
  62 = 'READ'
  78 = 's'
  121 = 'Start'
  36 = 'Stop'
  13 = 'Target Acceleration:'
  19 = 'Target Distance:'
  16 = 'Target Jerk:'
  12 = 'Target Speed:'
  35 = 'UP'
  91 = 'X:'
  81 = 'X增量'
  85 = 'X增量:'
  92 = 'Y:'
  82 = 'Y增量'
  84 = 'Y增量:'
  93 = 'Z:'
  83 = 'Z增量:'
  44 = '一号轴'
  41 = '使能电机'
  51 = '停止'
  71 = '全局速度:'
  70 = '全局速度值:'
  97 = '关节插补'
  99 = '关节规划'
  58 = '初始化A点'
  73 = '回零点'
  59 = '复位'
  79 = '外部位置:'
  42 = '失能电机'
  60 = '定零点'
  86 = '实时位置'
  87 = '实时坐标X:'
  88 = '实时坐标Y:'
  89 = '实时坐标Z:'
  94 = '平移增量'
  57 = '往复运动'
  75 = '执行'
  76 = '标记'
  56 = '标记A点'
  77 = '清零'
  53 = '状态'
  54 = '状态:'
  45 = '电机位置'
  50 = '电机位置:'
  46 = '电机速度'
  49 = '电机速度:'
  61 = '直线插补'
  80 = '直线规划'
  90 = '直线运动X增量:'
  96 = '笛卡尔规划'
  95 = '绝对位置'
  24 = '表格'
  98 = '规划'
  74 = '设定零点'
  63 = '读取CSV'
  72 = '读取外部位置'
  64 = '轴1设定值:'
  65 = '轴2设定值:'
  66 = '轴3设定值:'
  67 = '轴4设定值:'
  68 = '轴5设定值:'
  69 = '轴6设定值:'
  43 = '轴参数'
  100 = '轴数:%d'
  47 = '运动模式'
  48 = '运动模式:'
END_TEXTLIST

// ---- VISUs/Visualization.TcVIS
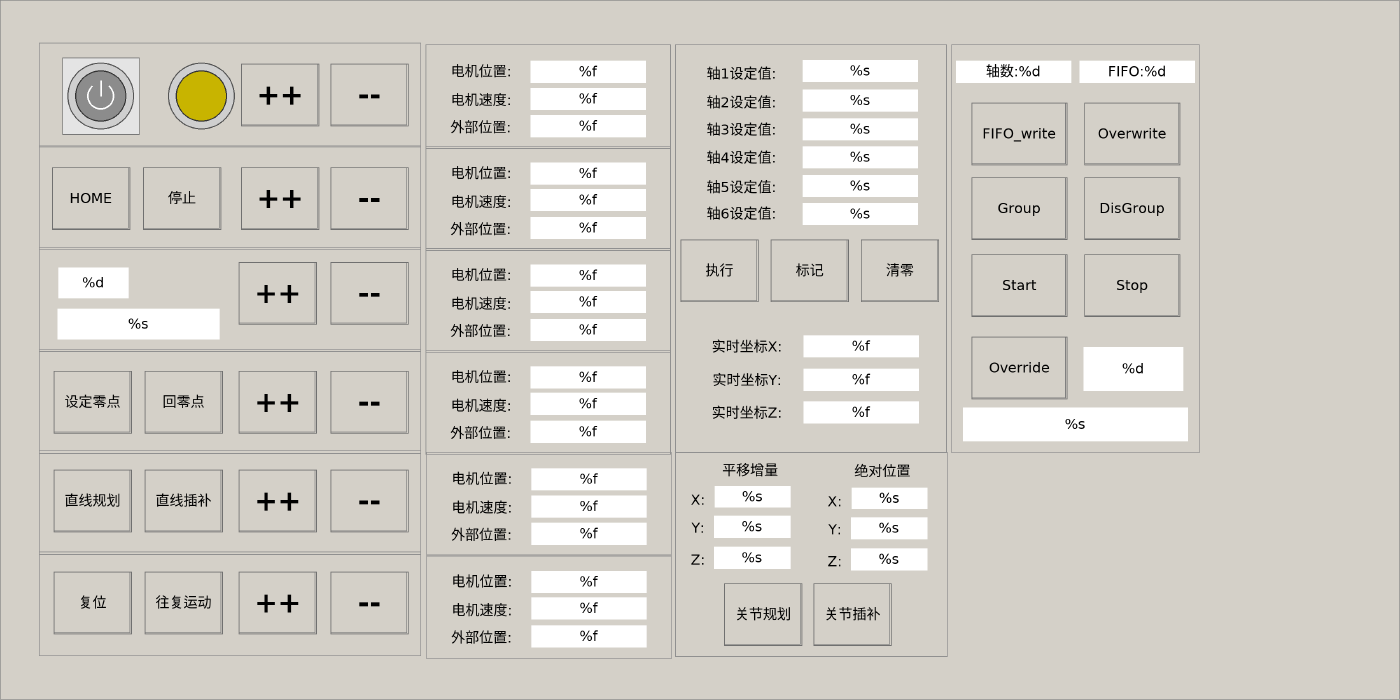
VISUALIZATION Visualization  // 1800x900
    GroupBox (50,47 491x142)
        Button (375,35 100x80), "--"
            OnMouseDown: execute { axisNum:=0; MAIN.CurrentJob:=4; }
            OnMouseUp: execute { axisNum:=0; MAIN.CurrentJob:=0; }
        Button (260,35 100x80), "++"
            OnMouseDown: execute { axisNum:=0; MAIN.CurrentJob:=3; }
            OnMouseUp: execute { axisNum:=0; MAIN.CurrentJob:=0; }
        PowerSwitch (17,27 125x99), variable: MAIN.POWER, behaviour: TOGGLE, style: Switch-PowerSwitch-Gray
        Lamp1 (134,27 150x99), variable: MAIN.LAMP, style: Lamp-Lamp1-Yellow
    GroupBox (547,49 315x142)
        Label (2,28 139x30), "电机位置:"
        Label (4,100 134x30), "外部位置:"
        Textfield (134,63 150x30), "%f", text variable: Axis[0].NcToPlc.ActVelo
        Textfield (134,28 150x30), "%f", text variable: Axis[0].NcToPlc.ActPos
        Textfield (134,98 150x30), "%f", text variable: ExtPos[0]
        Label (9,65 125x30), "电机速度:"
    GroupBox (547,180 315x142)
        Label (2,28 139x30), "电机位置:"
        Label (4,100 134x30), "外部位置:"
        Textfield (134,62 150x30), "%f", text variable: Axis[1].NcToPlc.ActVelo
        Textfield (134,28 150x30), "%f", text variable: Axis[1].NcToPlc.ActPos
        Textfield (134,98 150x30), "%f", text variable: ExtPos[1]
        Label (9,65 125x30), "电机速度:"
    GroupBox (547,311 315x142)
        Label (2,28 139x30), "电机位置:"
        Label (4,100 134x30), "外部位置:"
        Textfield (134,62 150x30), "%f", text variable: Axis[2].NcToPlc.ActVelo
        Textfield (134,28 150x30), "%f", text variable: Axis[2].NcToPlc.ActPos
        Textfield (134,98 150x30), "%f", text variable: ExtPos[2]
        Label (9,65 125x30), "电机速度:"
    GroupBox (547,442 315x142)
        Label (2,28 139x30), "电机位置:"
        Label (4,100 134x30), "外部位置:"
        Textfield (134,62 150x30), "%f", text variable: Axis[3].NcToPlc.ActVelo
        Textfield (134,28 150x30), "%f", text variable: Axis[3].NcToPlc.ActPos
        Textfield (134,98 150x30), "%f", text variable: ExtPos[3]
        Label (9,65 125x30), "电机速度:"
    GroupBox (548,573 315x142)
        Label (2,28 139x30), "电机位置:"
        Label (4,100 134x30), "外部位置:"
        Textfield (134,63 150x30), "%f", text variable: Axis[4].NcToPlc.ActVelo
        Textfield (134,28 150x30), "%f", text variable: Axis[4].NcToPlc.ActPos
        Textfield (134,98 150x30), "%f", text variable: ExtPos[4]
        Label (9,65 125x30), "电机速度:"
    GroupBox (50,179 491x142)
        Button (260,36 100x80), "++"
            OnMouseDown: execute { axisNum:=1; MAIN.CurrentJob:=3; }
            OnMouseUp: execute { axisNum:=1; MAIN.CurrentJob:=0; }
        Button (375,36 100x80), "--"
            OnMouseDown: execute { axisNum:=1; MAIN.CurrentJob:=4; }
            OnMouseUp: execute { axisNum:=1; MAIN.CurrentJob:=0; }
        Button (134,36 100x80), "停止"
            OnMouseClick: execute { MAIN.CurrentJob:=5; }
        Button (17,36 100x80), "HOME"
            OnMouseClick: execute { MAIN.CurrentJob:=6; }
    GroupBox (548,705 315x142)
        Label (2,28 139x30), "电机位置:"
        Label (4,100 134x30), "外部位置:"
        Textfield (134,62 150x30), "%f", text variable: Axis[5].NcToPlc.ActVelo
        Textfield (134,28 150x30), "%f", text variable: Axis[5].NcToPlc.ActPos
        Textfield (134,98 150x30), "%f", text variable: ExtPos[5]
        Label (9,65 125x30), "电机速度:"
    GroupBox (50,310 491x142)
        Button (257,27 100x80), "++"
            OnMouseDown: execute { axisNum:=2; MAIN.CurrentJob:=3; }
            OnMouseUp: execute { axisNum:=2; MAIN.CurrentJob:=0; }
        Button (375,27 100x80), "--"
            OnMouseDown: execute { axisNum:=2; MAIN.CurrentJob:=4; }
            OnMouseUp: execute { axisNum:=2; MAIN.CurrentJob:=0; }
        Textfield (24,33 92x41), "%d", text variable: MAIN.CurrentJob
        Textfield (23,86 210x41), "%s", text variable: MAIN.CurrentJobState
    GroupBox (50,441 491x142)
        Button (257,36 100x80), "++"
            OnMouseDown: execute { axisNum:=3; MAIN.CurrentJob:=3; }
            OnMouseUp: execute { axisNum:=3; MAIN.CurrentJob:=0; }
        Button (375,36 100x80), "--"
            OnMouseDown: execute { axisNum:=3; MAIN.CurrentJob:=4; }
            OnMouseUp: execute { axisNum:=3; MAIN.CurrentJob:=0; }
        Button (19,36 100x80), "设定零点"
            OnMouseClick: execute { MAIN.CurrentJob:=1; }
        Button (136,36 100x80), "回零点"
            OnMouseClick: execute { MAIN.CurrentJob:=11; }
    GroupBox (50,571 491x142)
        Button (257,33 100x80), "++"
            OnMouseDown: execute { axisNum:=4; MAIN.CurrentJob:=3; }
            OnMouseUp: execute { axisNum:=4; MAIN.CurrentJob:=0; }
        Button (375,33 100x80), "--"
            OnMouseDown: execute { axisNum:=4; MAIN.CurrentJob:=4; }
            OnMouseUp: execute { axisNum:=4; MAIN.CurrentJob:=0; }
        Button (19,33 100x80), "直线规划"
            OnMouseClick: execute { MAIN.CurrentJob:=10; }
        Button (136,33 100x80), "直线插补"
            OnMouseClick: execute { MAIN.CurrentJob:=2; }
    GroupBox (50,701 491x142)
        Button (257,34 100x80), "++"
            OnMouseDown: execute { axisNum:=5; MAIN.CurrentJob:=3; }
            OnMouseUp: execute { axisNum:=5; MAIN.CurrentJob:=0; }
        Button (375,34 100x80), "--"
            OnMouseDown: execute { axisNum:=5; MAIN.CurrentJob:=4; }
            OnMouseUp: execute { axisNum:=5; MAIN.CurrentJob:=0; }
        Button (19,34 100x80), "复位"
            OnMouseClick: execute {
                MAIN.CurrentJob:=9;
                //MoveA[0]:=-743179.666443;
                //MoveA[1]:=1499.826050;
                //MoveA[2]:=-1396.145325;
                //MoveA[3]:=6061.5802;
                //MoveA[4]:=1828.031616;
                //MoveA[5]:=-1145.742188;
            }
        Button (136,34 100x80), "往复运动"
            OnMouseClick: execute { MAIN.CurrentJob:=8; }
    GroupBox (868,49 349x533)
        Textfield (163,27 150x30), "%s", text variable: GVL.MoveAString[0]
            OnMouseClick: write MoveAString[0] via Edit
        Textfield (163,65 150x30), "%s", text variable: GVL.MoveAString[1]
            OnMouseClick: write MoveAString[1] via Edit
        Textfield (163,102 150x30), "%s", text variable: GVL.MoveAString[2]
            OnMouseClick: write MoveAString[2] via Edit
        Textfield (163,138 150x30), "%s", text variable: GVL.MoveAString[3]
            OnMouseClick: write MoveAString[3] via Edit
        Textfield (163,175 150x30), "%s", text variable: GVL.MoveAString[4]
            OnMouseClick: write MoveAString[4] via Edit
        Textfield (163,211 150x30), "%s", text variable: GVL.MoveAString[5]
            OnMouseClick: write MoveAString[5] via Edit
        Label (16,31 139x30), "轴1设定值:"
        Label (16,68 139x30), "轴2设定值:"
        Label (16,103 139x30), "轴3设定值:"
        Label (16,139 139x30), "轴4设定值:"
        Label (16,177 139x30), "轴5设定值:"
        Label (16,211 139x30), "轴6设定值:"
        Button (7,259 100x80), "执行"
            OnMouseClick: execute { MAIN.CurrentJob:=7; }
        Button (123,259 100x80), "标记"
            OnMouseClick: execute {
                MoveA[0]:=Axis[0].NcToPlc.ActPos;
                MoveA[1]:=Axis[1].NcToPlc.ActPos;
                MoveA[2]:=Axis[2].NcToPlc.ActPos;
                MoveA[3]:=Axis[3].NcToPlc.ActPos;
                MoveA[4]:=Axis[4].NcToPlc.ActPos;
                MoveA[5]:=Axis[5].NcToPlc.ActPos;
                MoveAString[0]:=LREAL_TO_STRING(MoveA[0]/24.995);
                MoveAString[1]:=LREAL_TO_STRING(MoveA[1]/32.28);
                MoveAString[2]:=LREAL_TO_STRING(MoveA[2]/49.845);
                MoveAString[3]:=LREAL_TO_STRING(MoveA[3]/50.905);
                MoveAString[4]:=LREAL_TO_STRING(MoveA[4]/80.34);
                MoveAString[5]:=LREAL_TO_STRING(MoveA[5]/60.5);
            }
        Label (23,382 139x30), "实时坐标X:"
        Textfield (164,381 150x30), "%f", text variable: Pos_Now[0]
        Textfield (164,424 150x30), "%f", text variable: Pos_Now[1]
        Textfield (164,466 150x30), "%f", text variable: Pos_Now[2]
        Button (239,259 100x80), "清零"
            OnMouseClick: execute {
                MoveA[0]:=0;
                MoveA[1]:=0;
                MoveA[2]:=0;
                MoveA[3]:=0;
                MoveA[4]:=0;
                MoveA[5]:=0;
                MoveAString[0]:='0';
                MoveAString[1]:='0';
                MoveAString[2]:='0';
                MoveAString[3]:='0';
                MoveAString[4]:='0';
                MoveAString[5]:='0';
            }
    Label (828,628 139x30), "X:"
    Label (828,664 139x30), "Y:"
    Label (828,705 139x30), "Z:"
    GroupBox (868,573 350x271)
        Label (136,57 139x30), "X:"
        Label (136,93 139x30), "Y:"
        Label (136,134 139x30), "Z:"
        Textfield (226,53 99x29), "%s", text variable: GVL.OutCMovePosString[0]
            OnMouseClick: write OutCMovePosString[0] via Edit
        Textfield (225,91 100x30), "%s", text variable: GVL.OutCMovePosString[1]
            OnMouseClick: write OutCMovePosString[1] via Edit
        Textfield (225,131 100x30), "%s", text variable: GVL.OutCMovePosString[2]
            OnMouseClick: write OutCMovePosString[2] via Edit
        Label (27,17 139x30), "平移增量"
        Label (197,18 139x30), "绝对位置"
        Button (63,177 100x80), "关节规划"
            OnMouseClick: execute { MAIN.CurrentJob:=13; }
        Button (178,177 100x80), "关节插补"
            OnMouseClick: execute { MAIN.CurrentJob:=12; }
    Label (891,474 139x30), "实时坐标Y:"
    Label (891,516 139x30), "实时坐标Z:"
    Textfield (918,624 99x29), "%s", text variable: GVL.OutMovePosString[0]
        OnMouseClick: write OutMovePosString[0] via Edit
    Textfield (917,662 100x30), "%s", text variable: GVL.OutMovePosString[1]
        OnMouseClick: write OutMovePosString[1] via Edit
    Textfield (917,702 100x30), "%s", text variable: GVL.OutMovePosString[2]
        OnMouseClick: write OutMovePosString[2] via Edit
    GroupBox (1223,49 319x533)
        Textfield (5,28 150x30), "轴数:%d", text variable: MAIN.FiFo_GetDimension.iNoOfAxes
        Textfield (164,28 150x30), "FIFO:%d", text variable: MAIN.FiFo_GetDimension.iNoOfFifoEntries
        Button (171,179 123x80), "DisGroup"
            tap MAIN.FiFo_GroupDisintegrate.bExecute
        Button (26,179 123x80), "Group"
            tap MAIN.integrate_do
        Button (26,278 123x80), "Start"
            tap MAIN.start_do
        Button (26,384 123x80), "Override"
            tap MAIN.FiFo_SetChannelOverride.bExecute
        Textfield (169,396 130x58), "%d", text variable: GVL.Axis[1].NcToPlc.SafEntries
        Button (26,83 123x80), "FIFO_write"
            tap MAIN.FIFO_write_do
        Button (171,83 123x80), "Overwrite"
            tap MAIN.FIFO_overwrite_do
        Textfield (14,474 291x45), "%s", text variable: MAIN.fifo_display
    Button (1394,327 123x80), "Stop"
        tap MAIN.stop_do
END_VISUALIZATION
